(*HEAT Ponics *)
(*
	IF ((Modbus.Balkon_temp > Modbus.Balkon_set_temp+1)   ) THEN
		HW_balkon_heat		:= FALSE;
	END_IF

	IF ((Modbus.Balkon_temp <  Modbus.Balkon_set_temp-1 ) ) THEN
		HW_balkon_heat		:=	TRUE;
	END_IF
*)
(*
pwm_par_balkon.bInstantPWMUpdate:=0;
pwm_par_balkon.tPWMPeriod:=T#5800ms;
pwm_par_balkon.tTaskCycleTime:=T#5ms;

pi_par_balkon.bARWOnIPartOnly:=0;
pi_par_balkon.fKp:=40;
pi_par_balkon.fOutMaxLimit:=100;
pi_par_balkon.fOutMinLimit:=0;
pi_par_balkon.tCtrlCycleTime:=T#5ms;
pi_par_balkon.tTaskCycleTime:=T#5ms;
pi_par_balkon.tTn:=T#30m;

pi_balkon(fSetpointValue:=Modbus.Balkon_set_temp, fActualValue :=Modbus.Balkon_temp, fManSyncValue :=0, bSync:=0, eMode:=2,bHold:=0, stParams:=pi_par_balkon, fOut => );
pwm_balkon(fPwmInput:=pi_balkon.fOut, eMode:=2, stParams:=pwm_par_balkon, bPwmOutBitPos=>HW_balkon_heat );
*)
END_PROGRAM

(* POU ExtractTime, ST *)
FUNCTION_BLOCK ExtractTime
VAR_INPUT
	tm:TOD;
END_VAR
VAR_OUTPUT
	h, m	: UINT;
END_VAR
VAR
	tw	: DWORD;

END_VAR
tw:=TOD_TO_DWORD(tm);
tw:=tw/(1000*60);
m:=DWORD_TO_UINT(tw MOD 60);
h:=DWORD_TO_UINT(tw / 60);
END_FUNCTION_BLOCK

(* POU Thermocontrol, ST *)
PROGRAM Thermocontrol
VAR
(*	period_sec		: INT:=120;  *)  (* Частота работы термостата, секунды*)
	gisterezis		: REAL:=0.2; (*Гистерезис термостата, градусы цельсия *)
	Timer1			: TON;
	Timer1Q			: BOOL;
	state			: INT:=0;
	 tTimerValue		: TIME:=t#120s;  (* Частота работы термостата, секунды*)
	pi_1f, pi_2f, pi_sauna 			: FB_CTRL_PI;
	pwm_1f, pwm_2f, pwm_sauna1	: FB_CTRL_PWM_OUT;

	pi_balkon 			: FB_CTRL_PI;
	pwm_balkon			: FB_CTRL_PWM_OUT;

	pi_septik				: FB_CTRL_PI;
	pwm_septik			: FB_CTRL_PWM_OUT;
	Power_septik			: UINT:=75;


END_VAR
(* tTimerValue := DINT_TO_TIME(period_sec*1000); *)

pwm_par_1f.bInstantPWMUpdate:=0;
pwm_par_1f.tPWMPeriod:=T#5135ms;
pwm_par_1f.tTaskCycleTime:=T#10ms;

pwm_par_2f.bInstantPWMUpdate:=0;
pwm_par_2f.tPWMPeriod:=T#5735ms;
pwm_par_2f.tTaskCycleTime:=T#10ms;


pwm_par_balkon.bInstantPWMUpdate:=0;
pwm_par_balkon.tPWMPeriod:=T#5800ms;
pwm_par_balkon.tTaskCycleTime:=T#10ms;
pi_par_balkon.bARWOnIPartOnly:=0;
pi_par_balkon.fKp:=40;
pi_par_balkon.fOutMaxLimit:=100;
pi_par_balkon.fOutMinLimit:=0;
pi_par_balkon.tCtrlCycleTime:=T#10ms;
pi_par_balkon.tTaskCycleTime:=T#10ms;
pi_par_balkon.tTn:=T#30m;

IF Modbus.Heat_pipe_septik_winter = TRUE THEN
	pwm_par_septik.bInstantPWMUpdate:=0;
	pwm_par_septik.tPWMPeriod:=T#15000ms;
	pwm_par_septik.tTaskCycleTime:=T#10ms;
	pwm_septik(fPwmInput:=Power_septik, eMode:=2, stParams:=pwm_par_septik, bPwmOutBitPos=>HW_septik_heat );

END_IF

(*
pi_par_septik.bARWOnIPartOnly:=0;
pi_par_septik.fKp:=40;
pi_par_septik.fOutMaxLimit:=100;
pi_par_septik.fOutMinLimit:=0;
pi_par_septik.tCtrlCycleTime:=T#5ms;
pi_par_septik.tTaskCycleTime:=T#5ms;
pi_par_septik.tTn:=T#30m;
*)





pi_balkon(fSetpointValue:=Modbus.Balkon_set_temp, fActualValue :=Modbus.Balkon_temp, fManSyncValue :=0, bSync:=0, eMode:=2,bHold:=0, stParams:=pi_par_balkon, fOut => );
pwm_balkon(fPwmInput:=pi_balkon.fOut, eMode:=2, stParams:=pwm_par_balkon, bPwmOutBitPos=>HW_balkon_heat );




pwm_par_sauna.bInstantPWMUpdate:=0;
pwm_par_sauna.tPWMPeriod:=T#300s;
pwm_par_sauna.tTaskCycleTime:=T#5ms;


pi_par_1f.bARWOnIPartOnly:=0;
pi_par_1f.fKp:=40;
pi_par_1f.fOutMaxLimit:=100;
pi_par_1f.fOutMinLimit:=0;
pi_par_1f.tCtrlCycleTime:=T#5ms;
pi_par_1f.tTaskCycleTime:=T#5ms;
pi_par_1f.tTn:=T#30m;

pi_par_sauna.bARWOnIPartOnly:=0;
pi_par_sauna.fKp:=40;
pi_par_sauna.fOutMaxLimit:=100;
pi_par_sauna.fOutMinLimit:=0;
pi_par_sauna.tCtrlCycleTime:=T#5ms;
pi_par_sauna.tTaskCycleTime:=T#5ms;
pi_par_sauna.tTn:=T#30m;

(**)
	pi_1f(fSetpointValue:=Modbus.First_floor_temp_target, fActualValue :=INT_TO_REAL(HW_temp_first_floor)/10, fManSyncValue :=0, bSync:=0, eMode:=2,bHold:=0, stParams:=pi_par_1f, fOut => );
(*	pi_1f(fSetpointValue:=Modbus.First_floor_temp_target, fActualValue :=Internal.First_floor_temp_SHT30, fManSyncValue :=0, bSync:=0, eMode:=2,bHold:=0, stParams:=pi_par_1f, fOut => );*)

	pwm_1f(fPwmInput:=pi_1f.fOut, eMode:=2, stParams:=pwm_par_1f, bPwmOutBitPos=>HW_heat_first_floor );

	pi_2f(fSetpointValue:=Modbus.Second_floor_temp_target, fActualValue :=INT_TO_REAL(HW_temp_second_floor)/10, fManSyncValue :=0, bSync:=0, eMode:=2,bHold:=0, stParams:=pi_par_1f, fOut => );
	pwm_2f(fPwmInput:=pi_2f.fOut, eMode:=2, stParams:=pwm_par_2f, bPwmOutBitPos=>HW_heat_second_floor );

(* SAUNA PID*)
(*
	pi_sauna(fSetpointValue:=Modbus.Sauna_temp_target, fActualValue :=INT_TO_REAL(HW_temp_sauna)/10, fManSyncValue :=0, bSync:=0, eMode:=2,bHold:=0, stParams:=pi_par_sauna, fOut => );
	pwm_sauna1(fPwmInput:=pi_sauna.fOut, eMode:=2, stParams:=pwm_par_sauna, bPwmOutBitPos=>HW_heat_Sauna );
*)

CASE state OF
0:
(*	IF (Modbus.First_floor_temp > Modbus.First_floor_temp_target+gisterezis ) THEN
		HW_heat_first_floor:=FALSE;
	END_IF

	IF ((Modbus.First_floor_temp <  Modbus.First_floor_temp_target-gisterezis) AND (Modbus.First_floor_temp <>0)  ) THEN
		HW_heat_first_floor:=TRUE;
	END_IF
*)

	state:=1;

1:
(*	IF (Modbus.Second_floor_temp > Modbus.Second_floor_temp_target+gisterezis ) THEN
		HW_heat_Second_floor:=FALSE;
	END_IF

	IF ((Modbus.Second_floor_temp <  Modbus.Second_floor_temp_target-gisterezis ) AND (Modbus.Second_floor_temp <>0)) THEN
		HW_heat_Second_floor:=TRUE;
	END_IF
*)
	state:=2;
2:
(* SAUNA GISTEREZIS *)

	IF (Modbus.Sauna_temp > Modbus.Sauna_temp_target+gisterezis ) THEN
		HW_heat_Sauna:=FALSE;
	END_IF

	IF ((Modbus.Sauna_temp <  Modbus.Sauna_temp_target-gisterezis ) AND (Modbus.Sauna_temp <>0)) THEN
		HW_heat_Sauna:=TRUE;
	END_IF
	state:=3;
3:


IF (Modbus.Sport_temp > Modbus.Sport_temp_target+gisterezis OR HW_heat_Sauna=TRUE ) THEN
		HW_heat_sport:=FALSE;
	END_IF

	IF ((Modbus.Sport_temp <  Modbus.Sport_temp_target-gisterezis ) AND (Modbus.Sport_temp <>0)  AND HW_heat_Sauna=FALSE) THEN
		HW_heat_sport:=TRUE;
	END_IF



	state:=4;

4:
	IF (Modbus.Underfloor_temp > Modbus.Underfloor_temp_target+gisterezis AND Modbus.Underfloor_hum < Modbus.Underfloor_humidity_target-1 ) THEN
		HW_heat_underfloor:=FALSE;
	END_IF

	IF ((Modbus.Underfloor_temp <  Modbus.Underfloor_temp_target-gisterezis OR Modbus.Underfloor_hum > Modbus.Underfloor_humidity_target+1) AND (Modbus.Underfloor_temp <>0)) THEN
		HW_heat_Underfloor:=TRUE;
	END_IF

	state:=100;



100:


	Timer1(IN:=NOT Timer1Q , PT:=tTimerValue , Q=>Timer1Q , ET=> );
		IF timer1.q THEN

		state:=0;
		END_IF



END_CASE
END_PROGRAM

(* POU Sensors, ST *)
PROGRAM Sensors
VAR
(*	Period_sensors_read		: INT:=30; *) (* Частота присвоения значений аналоговых температурных датчиков с модулей KL, секунды *)
	Timer					: TON;
	TimerQ					: BOOL;
	tTimerValue				: TIME:=t#30s; (* Частота присвоения значений аналоговых температурных датчиков с модулей KL, секунды *)
	Trigger_water_cold: F_TRIG;
	Water_count_house		: REAL;
	Water_count_teplica		: REAL;
END_VAR
Timer();
Trigger_water_cnt_impulse_teplica(CLK:=HW_I_rez5);

Trigger_water_cold(CLK :=HW_water_counter);
IF (Trigger_water_cold.Q) THEN

	(*Modbus.Kitchen_stat_cold_water:=Modbus.Kitchen_stat_cold_water+1; *)
	Water_count_house	:=	Water_count_house+1;
	Modbus.Sensor_house_water_imp	:=	Modbus.Sensor_house_water_imp+1;
END_IF

IF Trigger_water_cnt_impulse_teplica.Q THEN
	Water_count_teplica	:=	Water_count_teplica+1;
	Modbus.Teplica_cnt_water_pipe	:= 	Modbus.Teplica_cnt_water_pipe+1;
END_IF




(* tTimerValue := DINT_TO_TIME(Period_sensors_read*1000); *)

	Timer(IN:=NOT TimerQ , PT:=tTimerValue , Q=>TimerQ , ET=> );
	IF timer.q THEN

		Modbus.First_floor_temp		:=	INT_TO_REAL(HW_temp_first_floor)/10;
(*		Modbus.First_floor_temp		:=	Internal.First_floor_temp_SHT30; *)

		Modbus.Second_floor_temp	:=	INT_TO_REAL(HW_temp_second_floor)/10;
		Modbus.Sauna_temp			:=	INT_TO_REAL(HW_temp_sauna)/10;
		Modbus.Sport_temp			:=	INT_TO_REAL(HW_temp_sport)/10;

		Modbus.Underfloor_temp		:=	INT_TO_REAL(HW_temp_underfloor)/10;
(*		Modbus.Sport_underfloor_temp	:=	INT_TO_REAL(HW_temp_sport_underfloor)/10;	*)
		Modbus.Street_temp			:=	INT_TO_REAL(HW_temp_street)/10;
		Modbus.Vent_temp			:=	INT_TO_REAL(HW_temp_vent)/10;

		Modbus.Balkon_temp			:=	INT_TO_REAL(HW_temp_balkon)/10;
(*		Modbus.Drovnik_temp			:=	INT_TO_REAL(HW_temp_drovnik)/10;
		Modbus.Sklad_temp			:= 	INT_TO_REAL(HW_temp_sklad)/10;	*)

	END_IF
END_PROGRAM

(* POU Security_new, ST *)
PROGRAM Security_new
VAR
(*	TRIG_PIR_terrasa			:	F_TRIG;
	TRIG_PIR_zapad			:	F_TRIG;
	TRIG_PIR_vostok			:	F_TRIG;
	TRIG_PIR_sport			:	F_TRIG;
	TRIG_GERKON_drovnik	:	F_TRIG;
	TRIG_sensor_smoke_1floor:	F_TRIG;

	trig_mem_terrasa				:	BOOL:=FALSE;
	trig_mem_zapad				:	BOOL:=FALSE;
	trig_mem_vostok				:	BOOL:=FALSE;
	trig_mem_sport				:	BOOL:=FALSE;
	trig_mem_drovnik				:	BOOL:=FALSE;
	trig_mem_sensor_smoke_1floor	:	BOOL:=FALSE;
*)
END_VAR
iobroker.PIR_terrasa			 :=HW_PIR_terrasa;
iobroker.PIR_zapad			 :=HW_PIR_zapad;
iobroker.PIR_vostok 			 :=HW_PIR_vostok;
iobroker.PIR_sport			 :=HW_PIR_sport;
iobroker.GERKON_drovnik		 :=HW_GERKON_drovnik;
(*
Modbus.Smoke_1floor				 :=HW_sensor_smoke_1floor;
Modbus.Smoke_2floor			 	:=HW_sensor_smoke_2floor;
Modbus.Smoke_sport				 :=HW_sensor_smoke_sport;
Modbus.Smoke_sklad				 :=HW_sensor_smoke_sklad;
Modbus.Smoke_drovnik			 :=HW_sensor_smoke_drovnik;
*)

Modbus.PIR_terrasa			 :=HW_PIR_terrasa;
Modbus.PIR_zapad			 :=HW_PIR_zapad;
Modbus.PIR_vostok 			 :=HW_PIR_vostok;
Modbus.PIR_sport				 :=HW_PIR_sport;
Modbus.PIR_north_zapad		 :=HW_PIR_north_zapad;
Modbus.PIR_north_vostok		 :=HW_PIR_north_vostok;

Modbus.GERKON_door		 :=HW_GERKON_door;
Modbus.GERKON_drovnik		 :=HW_GERKON_drovnik;
Modbus.GERKON_sklad		 :=HW_GERKON_sklad;



(* Modbus.Smoke				 :=HW_sensor_smoke_1floor; *)
END_PROGRAM

(* POU RS485read, ST *)
PROGRAM RS485read
VAR

	tTimerValue				: TIME	:=	t#60s; (* Период опроса RS485*)
	FtrigBusy				: F_TRIG;
	timeoutvalue				: TIME := T#2000ms;		(* timeout while waiting for an answer of the modbus slave *)
	state					: INT;
	busy					: BOOL;
	LastErrorstate				: INT;
	LastModbusError			: ST_ModbusErrorDiagnostics;
	CounterError				: DINT;
	CounterSuccess			: DINT;
	i,k,l						: INT:=1;

	teplica_ADM4188_id			: BYTE:=16#45;
	klubnika_WP8025ADAM		: BYTE:=16#46;
	klubnika_SHT30				: BYTE:=16#64;


	sensors_SHT20_v1_id			: ARRAY[1..3] OF BYTE:= 16#0F, 16#05, 16#36;
	sensors_SHT20_v1_hum		: ARRAY[1..3] OF REAL:=3(0);
	sensors_SHT20_v1_temp		: ARRAY[1..3] OF REAL:=3(0);

(*	sensors_SHT20_v2_id			: ARRAY[1..1] OF BYTE:=  16#0A; *)
	sensors_SHT20_v2_id			: ARRAY[1..1] OF BYTE:=  16#35;

	sensors_SHT20_v2_hum		: ARRAY[1..1] OF REAL:=1(0);
	sensors_SHT20_v2_temp		: ARRAY[1..1] OF REAL:=1(0);


	sensors_SHT30_v3_id			: ARRAY[1..8] OF BYTE:= 16#14, 16#11,16#29, 16#30,16#07,16#08, 16#32, 16#35;
	sensors_SHT30_v3_hum		: ARRAY[1..8] OF REAL:=8(0);
	sensors_SHT30_v3_temp		: ARRAY[1..8] OF REAL:=8(0);

	sensors_CO2_id				: ARRAY[1..4] OF BYTE:=16#68, 16#69,16#6A, 16#6B ;
	sensors_CO2_ppm			: ARRAY[1..4] OF INT;

	house_DS18B20_id			: BYTE:=16#64;
	sensors_DS18B20_temp		: ARRAY[1..8] OF REAL:=8(0);
	parnik_DS18B20_id			: BYTE:=16#64;
	teplica_DS18B20_temp		: ARRAY[1..8] OF REAL:=8(0);
	teplica_gate_pt1000_id			: BYTE:=70;
	MBdata8_pt1000				 : ARRAY [1..8] OF INT;
	MBdata_teplica_gate_pt1000	: ARRAY [1..8] OF REAL;

	MBdata						 : ARRAY [1..2] OF INT;
	MBdata8						 : ARRAY [1..8] OF UINT;
	MBdata8_h					 : ARRAY [1..8] OF UINT;

	sensor_ponics_PH_id			: BYTE:= 16#4F ;
	sensor_teplica_PH_id			: BYTE:= 16#78 ;
	MBdata_sensor_ponics_PH	: ARRAY [1..4] OF INT;
	MBdata_sensor_teplica_PH	: ARRAY [1..4] OF INT;

	Teplica_tank_level_id			: BYTE:=1;
	Teplica_tankA_level_id		: BYTE:=2;
	Teplica_tankB_level_id		: BYTE:=3;

	Teplica_ph_sensor_low		: REAL;
	Teplica_ph_sensor_temp		: REAL;
	Teplica_ph_sensor_mv		: REAL;
(*	Teplica_temp_air				: REAL; *)
	Teplica_temp_pip_heat_in		: REAL;

	Ponics_ph_sensor_mv			: REAL;

	sensor_teplica_EC_id			: BYTE:= 16#C8 ;
	sensor_ponics_EC_id			: BYTE:= 16#51 ;
	sensor_ponics_EC2_id			: BYTE:= 16#50 ;
	sensor_ponics_EC_int			: INT;
	sensor_ponics_EC2_int		: INT;
	MBdata_sensor_teplica_EC		 : ARRAY [1..4] OF INT;
	MBdata_sensor_ponics_EC2	 :  INT;

	balkon_light_sensor_id			: BYTE:=16#5A;
	balkon_light_word2			: WORD;
	teplica_light_sensor_id			: BYTE:=16#3C;
	teplica_light_low				: WORD;
	teplica_light_high				: WORD;
	teplica_light_dword			: DWORD;
	teplica_light_array				: ARRAY [1..2] OF WORD;

	password_1				: ARRAY [1..6] OF BYTE:=6(1); (* пароль к меркуриям, по умолчанию 6 единиц*)
	crctest					: WORD;
	get_energy_E_T1			: FB_GET_ENERGY;
	get_energy_E_T2			: FB_GET_ENERGY;
	get_energy_MT			: FB_GET_ENERGY;
	get_supply				: FB_GET_SUPPLY;
	get_current				: FB_GET_CURRENT;
	get_power				: FB_GET_POWER;
	energyMT					: ARRAY[1..12,1..2] OF REAL;
	get_current_done			: BOOL;
	get_power_done			: BOOL;
	get_energy_E_T1_done	: BOOL;
	get_energy_E_T2_done	: BOOL;
	get_energy_MT_done		: BOOL;
	get_supply_done			: BOOL;
	arrReceive				: ARRAY[1..5] OF BYTE;
	arrSend					: ARRAY[1..5] OF BYTE;
	t,m, tr, none				: INT:=1;
	 e_rs1					: INT:=0;
	ponics_EC2_1				: REAL;
	ponics_EC2_2				: REAL;
	ponics_EC2_3				: REAL;
	ponics_EC2_4				: REAL;
	Modbus_errors			:DWORD;
	Modbus_array_errors		:ARRAY[0..254] OF BYTE;
	Balkon_CO2				: INT;
	Teplica_CO2				: INT;
	Timer_wait_RS			: TON;
	 tTimerValue_wait_RS1		: TIME:=t#2s;  (* *)
	cnt_err_read_tank			:UDINT;
	cnt_err_read_all			:UDINT;
	Temp_water_tank_DS		: REAL;
	Teplica_temp_panel		: REAL;
	teplica_tank_level_word	: ARRAY[0..17] OF WORD;
	teplica_tankA_level_word	: ARRAY[0..17] OF WORD;
	teplica_tankB_level_word	: ARRAY[0..17] OF WORD;

	Teplica_tank_level		: REAL;
	Teplica_tankA_level		: REAL;
	Teplica_tankB_level		: REAL;

	cnt_clear_di_2: BOOL;
	zero						: INT:=0;
	MBdataDI		 			 : ARRAY [1..8] OF UINT;
	Teplica_DO1			:	BOOL;
	Teplica_DO2			:	BOOL;
	Teplica_DO3			:	BOOL;
	Teplica_DO4			:	BOOL;
	Teplica_DO5			:	BOOL;
	Teplica_DO6			:	BOOL;
	Teplica_DO7			:	BOOL;
	Teplica_DO8			:	BOOL;

	MBdataDO_byte: BYTE;
	MBdataDO_byte_read: BYTE;
	test: BOOL;
END_VAR
(*Modbus.RS485_1_cnt_error		:= Modbus.RS485_1_cnt_error;
Modbus.RS485_1_cnt_success	:= Modbus.RS485_1_cnt_success;
*)

MBdataDO_byte.0			:=	Modbus.Teplica_pomp_fertA;
MBdataDO_byte.1			:=	Modbus.Teplica_pomp_fertB;
MBdataDO_byte.2			:=	Modbus.Teplica_zone_poliv;
MBdataDO_byte.3			:=	Modbus.Teplica_window_opener;
MBdataDO_byte.4			:=	Modbus.Teplica_pomp_cold;
MBdataDO_byte.5			:=	Modbus.Teplica_tank_heat;
MBdataDO_byte.7			:= 	Modbus.Light_garden;

CASE state OF
0:
		MB.ReadRegs(Execute:= FALSE);
		state := 2;

		e_rs1	:=0;
		Modbus_array_errors[0] :=0;
		Modbus_array_errors[1] :=0;
		Modbus_array_errors[2] :=0;
		Modbus_array_errors[3] :=0;
		Modbus_array_errors[4] :=0;
		Modbus_array_errors[5] :=0;
		Modbus_array_errors[6] :=0;
		Modbus_array_errors[7] :=0;
		Modbus_array_errors[8] :=0;
		Modbus_array_errors[9] :=0;
		Modbus_array_errors[10] :=0;



1:

		MB.ReadInputRegs(
			UnitID:= sensors_SHT20_v2_id[l],
			Quantity:= 2,
			MBAddr:= 512,
			cbLength:= 4,
			pMemoryAddr:= ADR(MBdata),
			Execute:= TRUE,
			Timeout:= timeoutvalue,
			Busy => busy,
		);
		IF NOT busy THEN
			IF (mb.Error = FALSE ) THEN
				sensors_SHT20_v2_temp[l]:=INT_TO_REAL(MBdata[1])/10;
				sensors_SHT20_v2_hum[l]:=INT_TO_REAL(MBdata[2])/10;
			ELSE
				Modbus_array_errors[e_rs1]	:= sensors_SHT20_v2_id[l];
				e_rs1	:= e_rs1+1;
			END_IF

			l:=l+1;
			MB.ReadRegs(Execute:= FALSE);
			IF (l>1 )	THEN
				l:=1;
				Modbus.Balkon_hum	:=	sensors_SHT20_v2_hum[1];

(*				Internal.Sport_underfloor_temp_SHT20		:=	sensors_SHT20_v2_temp[1];
				Internal.Sport_underfloor_hum				:=	sensors_SHT20_v2_hum[1];


				Modbus.Sport_underfloor_temp_SHT20		:=	(sensors_SHT20_v2_temp[1]);
				Modbus.Sport_underfloor_hum				:=	(sensors_SHT20_v2_hum[1]);
*)
				state :=2;
			ELSE
				state :=1;
			END_IF

		END_IF



2:
		MB.ReadRegs(
			UnitID:= sensors_SHT20_v1_id[i],
			Quantity:= 2,
			MBAddr:= 0,
			cbLength:= 4,
			pMemoryAddr:= ADR(MBdata),
			Execute:= TRUE,
			Timeout:= timeoutvalue,
			Busy => busy,
		);
		IF NOT busy THEN
			IF (mb.Error = FALSE ) THEN
				sensors_SHT20_v1_temp[i]:=INT_TO_REAL(MBdata[1])/10;
				sensors_SHT20_v1_hum[i]:=INT_TO_REAL(MBdata[2])/10;
			ELSE
				Modbus_array_errors[e_rs1]	:= sensors_SHT20_v1_id[i];

				e_rs1	:= e_rs1+1;
			END_IF
			i:=i+1;
			MB.ReadRegs(Execute:= FALSE);
			IF (i>3 )	THEN
				i:=1;
				Internal.Street_temp_SHT20			:=	sensors_SHT20_v1_temp[1];
				Internal.Street_hum				:=	sensors_SHT20_v1_hum[1];
				Internal.Sklad_temp_SHT20			:=	sensors_SHT20_v1_temp[2];
				Internal.Sklad_hum				:=	sensors_SHT20_v1_hum[2];

				Modbus.Street_temp_SHT20		:=	sensors_SHT20_v1_temp[1];
				Modbus.Street_hum				:=	sensors_SHT20_v1_hum[1];
				Modbus.Sklad_temp_SHT20		:=	sensors_SHT20_v1_temp[2];
				Modbus.Sklad_hum				:=	sensors_SHT20_v1_hum[2];
				Modbus.Parnik_sht_air_temp		:=	(sensors_SHT20_v1_temp[3])/10;
				Modbus.Parnik_sht_air_hum		:=	(sensors_SHT20_v1_hum[3])/10;
				state :=3;
			ELSE
				state :=2;
			END_IF

		END_IF


3:
		MB.ReadRegs(
			UnitID:= sensors_SHT30_v3_id[i],
			Quantity:= 2,
			MBAddr:= 512,
			cbLength:= 4,
			pMemoryAddr:= ADR(MBdata),
			Execute:= TRUE,
			Timeout:= timeoutvalue,
			Busy => busy,
		);
		IF NOT busy THEN
			IF (mb.Error = FALSE ) THEN
				sensors_SHT30_v3_temp[i]:=INT_TO_REAL(MBdata[1])/10;
				sensors_SHT30_v3_hum[i]:=INT_TO_REAL(MBdata[2])/10;
			ELSE
				Modbus_array_errors[e_rs1]	:= sensors_SHT30_v3_id[i];

				e_rs1	:= e_rs1+1;
			END_IF
			i:=i+1;
			MB.ReadRegs(Execute:= FALSE);
			IF (i>8 )	THEN
				i:=1;
				Internal.Drovnik_temp_SHT30		:=	sensors_SHT30_v3_temp[1];
				Internal.Drovnik_hum				:=	sensors_SHT30_v3_hum[1];
				Internal.Sport_temp_SHT30			:=	sensors_SHT30_v3_temp[2];
				Internal.Sport_hum					:=	sensors_SHT30_v3_hum[2];
				Internal.First_floor_temp_SHT30		:=	sensors_SHT30_v3_temp[3];
				Internal.First_floor_hum				:=	sensors_SHT30_v3_hum[3];
				Internal.Second_floor_temp_SHT30	:=	sensors_SHT30_v3_temp[4];
				Internal.Second_floor_hum			:=	sensors_SHT30_v3_hum[4];
				Internal.Underfloor_temp_SHT30		:=	sensors_SHT30_v3_temp[5];
				Internal.Underfloor_hum			:=	sensors_SHT30_v3_hum[5];
				Internal.Sport_underfloor_temp_SHT30		:=	sensors_SHT30_v3_temp[6];
				Internal.Sport_underfloor_hum				:=	sensors_SHT30_v3_hum[6];
				Internal.Teplica_temp_SHT30		:=	sensors_SHT30_v3_temp[7];
				Internal.Teplica_hum_SHT30		:=	sensors_SHT30_v3_hum[7];

				Modbus.Drovnik_temp_SHT30		:=	sensors_SHT30_v3_temp[1];
				Modbus.Drovnik_hum				:=	sensors_SHT30_v3_hum[1];
				Modbus.Sport_temp_SHT30		:=	sensors_SHT30_v3_temp[2];
				Modbus.Sport_hum				:=	sensors_SHT30_v3_hum[2];
				Modbus.First_floor_temp_SHT30	:=	sensors_SHT30_v3_temp[3];
				Modbus.First_floor_hum			:=	sensors_SHT30_v3_hum[3];
				Modbus.Second_floor_temp_SHT30	:=	sensors_SHT30_v3_temp[4];
				Modbus.Second_floor_hum			:=	sensors_SHT30_v3_hum[4];
				Modbus.Underfloor_temp_SHT30	:=	sensors_SHT30_v3_temp[5];
				Modbus.Underfloor_hum			:=	sensors_SHT30_v3_hum[5];
				Modbus.Sport_underfloor_temp_SHT30		:=	(sensors_SHT30_v3_temp[6]);
				Modbus.Sport_underfloor_hum				:=	(sensors_SHT30_v3_hum[6]);
				Modbus.Teplica_temp_SHT30		:=	sensors_SHT30_v3_temp[7];
				Modbus.Teplica_temp_air			:=	sensors_SHT30_v3_temp[7];
				Modbus.Teplica_hum_SHT30		:=	sensors_SHT30_v3_hum[7];
				Modbus.Balkon_hum				:=	sensors_SHT30_v3_hum[8];
				state :=4;
			ELSE
				state :=3;
			END_IF

		END_IF

4:
		MB.ReadInputRegs(
			UnitID:=sensors_CO2_id[k], (* station address *)
			Quantity:= 1,
			MBAddr:= 3,
			cbLength:= 2,
			pMemoryAddr:= ADR(MBdata),
			Execute:= TRUE,
			Timeout:= timeoutvalue,
			Busy => busy	);
		IF NOT busy THEN
			IF (mb.Error = FALSE ) THEN
				sensors_CO2_ppm[k]	:=	(MBdata[1]);
			ELSE
				Modbus_array_errors[e_rs1]	:= sensors_CO2_id[k];
				e_rs1	:= e_rs1+1;
			END_IF
			k:=k+1;
			MB.ReadRegs(Execute:= FALSE);
			IF (k>4 )	THEN
				k:=1;
				Modbus.Second_floor_CO2		:=	(sensors_CO2_ppm[1]);
				Modbus.First_floor_CO2		:=	(sensors_CO2_ppm[2]);
				Modbus.Balkon_CO2			:=	(sensors_CO2_ppm[3]);
				Modbus.Teplica_CO2			:=	(sensors_CO2_ppm[4]);

				state :=6;
			ELSE
				state :=4;
			END_IF
		END_IF




5:

		MB.ReadRegs(
			UnitID:= house_DS18B20_id,
			Quantity:= 8,
			MBAddr:= 0,
			cbLength:= 16,
			pMemoryAddr:= ADR(MBdata8_h),
			Execute:= TRUE,
			Timeout:= timeoutvalue,
			Busy => busy,
		);
		IF NOT busy THEN
			IF (mb.Error = FALSE ) THEN
(*				sensors_DS18B20_temp[1]:=INT_TO_REAL(MBdata8_h[1])/10;
				sensors_DS18B20_temp[2]:=INT_TO_REAL(MBdata8_h[2])/10;
				sensors_DS18B20_temp[3]:=INT_TO_REAL(MBdata8_h[3])/10;
				sensors_DS18B20_temp[4]:=INT_TO_REAL(MBdata8_h[4])/10;
*)
				IF (MBdata8_h[1] < 10000)
					THEN	sensors_DS18B20_temp[1]:=UINT_TO_REAL(MBdata8_h[1])/10;
				ELSE
					sensors_DS18B20_temp[1]:=-1*UINT_TO_REAL(MBdata8_h[1]-10000)/10;
				END_IF

				IF (MBdata8_h[2] < 10000)
					THEN	sensors_DS18B20_temp[2]:=UINT_TO_REAL(MBdata8_h[2])/10;
				ELSE
					sensors_DS18B20_temp[2]:=-1*UINT_TO_REAL(MBdata8_h[2]-10000)/10;
				END_IF


				IF (MBdata8_h[3] < 10000)
					THEN	sensors_DS18B20_temp[3]:=UINT_TO_REAL(MBdata8_h[3])/10;
				ELSE
					sensors_DS18B20_temp[3]:=-1*UINT_TO_REAL(MBdata8_h[3]-10000)/10;
				END_IF

				IF (MBdata8_h[5] < 10000)
					THEN	sensors_DS18B20_temp[5]:=UINT_TO_REAL(MBdata8_h[5])/10;
				ELSE
					sensors_DS18B20_temp[5]:=-1*UINT_TO_REAL(MBdata8_h[5]-10000)/10;
				END_IF



				IF  (sensors_DS18B20_temp[5] <>0 AND sensors_DS18B20_temp[5] <>85)	THEN
					Modbus.Rezerv_temp			:=	sensors_DS18B20_temp[5];
				END_IF
(*
				IF  (sensors_DS18B20_temp[2] <>0 AND sensors_DS18B20_temp[2] <>85)	THEN
					Modbus.		:=	sensors_DS18B20_temp[2];
				END_IF

				IF  (sensors_DS18B20_temp[3] <>0 AND sensors_DS18B20_temp[3] <>85)	THEN
					Modbus. 	:=	sensors_DS18B20_temp[3];
				END_IF

				IF  (sensors_DS18B20_temp[4] <>0 AND sensors_DS18B20_temp[4] <>85)	THEN
					Modbus. 	:=	sensors_DS18B20_temp[4];
				END_IF
*)

			ELSE
				Modbus_array_errors[e_rs1]	:= house_DS18B20_id;
				e_rs1	:= e_rs1+1;
			END_IF
			MB.ReadRegs(Execute:= FALSE);
			state:=6;

		END_IF


6:

		MB.ReadRegs(
			UnitID:= parnik_DS18B20_id,
			Quantity:= 8,
			MBAddr:= 0,
			cbLength:= 16,
			pMemoryAddr:= ADR(MBdata8),
			Execute:= TRUE,
			Timeout:=  T#2000ms,
			Busy => busy,
		);
		IF NOT busy THEN
			IF (MB.Error = FALSE ) THEN
				IF (MBdata8[1] < 10000)
					THEN	teplica_DS18B20_temp[1]:=UINT_TO_REAL(MBdata8[1])/10;
				ELSE
					teplica_DS18B20_temp[1]:=-1*UINT_TO_REAL(MBdata8[1]-10000)/10;
				END_IF

				IF (MBdata8[2] < 10000)
					THEN	teplica_DS18B20_temp[2]:=UINT_TO_REAL(MBdata8[2])/10;
				ELSE
					teplica_DS18B20_temp[2]:=-1*UINT_TO_REAL(MBdata8[2]-10000)/10;
				END_IF


				IF (MBdata8[3] < 10000)
					THEN	teplica_DS18B20_temp[3]:=UINT_TO_REAL(MBdata8[3])/10;
				ELSE
					teplica_DS18B20_temp[3]:=-1*UINT_TO_REAL(MBdata8[3]-10000)/10;
				END_IF

				IF (MBdata8[4] < 10000)
					THEN	teplica_DS18B20_temp[4]:=UINT_TO_REAL(MBdata8[4])/10;
				ELSE
					teplica_DS18B20_temp[4]:=-1*UINT_TO_REAL(MBdata8[4]-10000)/10;
				END_IF

				IF (MBdata8[5] < 10000)
					THEN	teplica_DS18B20_temp[5]:=UINT_TO_REAL(MBdata8[5])/10;
				ELSE
					teplica_DS18B20_temp[5]:=-1*UINT_TO_REAL(MBdata8[5]-10000)/10;
				END_IF


				IF  (teplica_DS18B20_temp[1] <>0 AND teplica_DS18B20_temp[1] <>85 AND teplica_DS18B20_temp[1] > -60  )	THEN
					Modbus.Parnik_air_temp	:= 		teplica_DS18B20_temp[1];
				END_IF

				IF  (teplica_DS18B20_temp[2] <>0 AND teplica_DS18B20_temp[2] <>85 AND teplica_DS18B20_temp[2] > -60)	THEN
					Modbus.Parnik_ground_temp		:=	teplica_DS18B20_temp[2];
				END_IF


				IF  (teplica_DS18B20_temp[3] <>0 AND teplica_DS18B20_temp[3] <>85  AND teplica_DS18B20_temp[3] > -60)	THEN
					Modbus.Parnik_pipe_temp	 	:=	teplica_DS18B20_temp[3];
				END_IF

(*				IF  (teplica_DS18B20_temp[4] <>0 AND teplica_DS18B20_temp[4] <>85 AND teplica_DS18B20_temp[4] > -60)	THEN

					Temp_water_tank_DS				:=	teplica_DS18B20_temp[4];
				END_IF

				IF  (teplica_DS18B20_temp[5] <>0 AND teplica_DS18B20_temp[5] <>85 AND teplica_DS18B20_temp[5] > -60)	THEN
					Teplica_temp_pip_heat_in 	:=	teplica_DS18B20_temp[5];
				END_IF

				IF  (teplica_DS18B20_temp[1]  = 0 OR teplica_DS18B20_temp[2]  = 0 OR teplica_DS18B20_temp[3]  = 0 OR teplica_DS18B20_temp[4]  = 0OR  teplica_DS18B20_temp[5]  = 0) THEN
					cnt_err_read_all	:=	cnt_err_read_all+1;
				END_IF

*)


			ELSE
				Modbus_array_errors[e_rs1]	:= parnik_DS18B20_id;
				e_rs1	:= e_rs1+1;
			END_IF
			MB.ReadRegs(Execute:= FALSE);
				state:=7;

		END_IF




7:

		MB.ReadRegs(
			UnitID:= balkon_light_sensor_id,
			Quantity:= 1,
			MBAddr:= 6,
			cbLength:= 2,
			pMemoryAddr:= ADR(balkon_light_word2),
			Execute:= TRUE,
			Timeout:= timeoutvalue,
			Busy => busy,
		);
		IF NOT busy THEN
			IF (mb.Error = FALSE ) THEN
				Modbus.Balkon_light_lux		:=	WORD_TO_UDINT(balkon_light_word2);
			ELSE
				Modbus_array_errors[e_rs1]	:= balkon_light_sensor_id;
				e_rs1	:= e_rs1+1;
			END_IF
			MB.ReadRegs(Execute:= FALSE);
			state:=8;
		END_IF

8:

		MB.ReadRegs(
			UnitID:= teplica_light_sensor_id,
			Quantity:= 2,
			MBAddr:= 2,
			cbLength:= 4,
			pMemoryAddr:= ADR(teplica_light_array),
			Execute:= TRUE,
			Timeout:= timeoutvalue,
			Busy => busy,
		);
		IF NOT busy THEN
			IF (MB.Error = FALSE ) THEN
				teplica_light_high:=teplica_light_array[1];
				teplica_light_low:=teplica_light_array[2];
				teplica_light_dword:=(teplica_light_array[1]*65535)+teplica_light_array[2];
				Modbus.Teplica_light_lux		:=	DWORD_TO_REAL(teplica_light_dword);


			ELSE
				Modbus_array_errors[e_rs1]	:= teplica_light_sensor_id;
				e_rs1	:= e_rs1+1;
			END_IF
			MB.ReadRegs(Execute:= FALSE);
			state:=9;
		END_IF

9:

		MB.ReadRegs(
			UnitID:= sensor_ponics_PH_id,
			Quantity:= 4,
			MBAddr:= 0,
			cbLength:= 8,
			pMemoryAddr:= ADR(MBdata_sensor_ponics_PH),
			Execute:= TRUE,
			Timeout:= timeoutvalue,
			Busy => busy,
		);
		IF NOT busy THEN
			IF (mb.Error = FALSE ) THEN
				Modbus.Ponics_PH			:=	INT_TO_REAL(MBdata_sensor_ponics_PH[1])/100;
				Modbus.Ponics_tank_temp		:=	INT_TO_REAL(MBdata_sensor_ponics_PH[3])/10;
				Ponics_ph_sensor_mv			:=	INT_TO_REAL(MBdata_sensor_ponics_PH[4]);

			ELSE
				Modbus_array_errors[e_rs1]	:= sensor_ponics_PH_id;
				e_rs1	:= e_rs1+1;

			END_IF
			MB.ReadRegs(Execute:= FALSE);
			state:=11;
		END_IF

10:

		MB.ReadRegs(
			UnitID:= sensor_teplica_PH_id,
			Quantity:= 4,
			MBAddr:= 0,
			cbLength:= 8,
			pMemoryAddr:= ADR(MBdata_sensor_teplica_PH),
			Execute:= TRUE,
			Timeout:= timeoutvalue,
			Busy => busy,
		);
		IF NOT busy THEN
			IF (MB.Error = FALSE ) THEN
				Modbus.Teplica_sensor_soil_PH	:=	INT_TO_REAL(MBdata_sensor_teplica_PH[1])/100;
				Teplica_ph_sensor_low			:=	INT_TO_REAL(MBdata_sensor_teplica_PH[2])/10;
				Teplica_ph_sensor_temp			:=	INT_TO_REAL(MBdata_sensor_teplica_PH[3])/10;
				Teplica_ph_sensor_mv			:=	INT_TO_REAL(MBdata_sensor_teplica_PH[4]);

			ELSE
				Modbus_array_errors[e_rs1]	:= sensor_teplica_PH_id;
				e_rs1	:= e_rs1+1;

			END_IF
			MB.ReadRegs(Execute:= FALSE);
			state:=11;
		END_IF


11:

		MB.ReadRegs(
			UnitID:= sensor_ponics_EC_id,
			Quantity:= 1,
			MBAddr:= 2,
			cbLength:= 2,
			pMemoryAddr:= ADR(sensor_ponics_EC_int),
			Execute:= TRUE,
			Timeout:= timeoutvalue,
			Busy => busy,
		);
		IF NOT busy THEN
			IF (mb.Error = FALSE ) THEN
			Modbus.Ponics_EC	:=	 INT_TO_REAL(sensor_ponics_EC_int)/1000;
				IF(Modbus.Ponics_EC < 0)	THEN
					Modbus.Ponics_EC	:= 0;
				END_IF
			ELSE
				Modbus_array_errors[e_rs1]	:= sensor_ponics_EC_id;
				e_rs1	:= e_rs1+1;
			END_IF
			MB.ReadRegs(Execute:= FALSE);
			state:=12;
		END_IF

12:

		MB.ReadRegs(
			UnitID:= sensor_teplica_EC_id,
			Quantity:= 4,
			MBAddr:= 0,
			cbLength:= 8,
			pMemoryAddr:= ADR(MBdata_sensor_teplica_EC),
			Execute:= TRUE,
			Timeout:= timeoutvalue,
			Busy => busy,
		);
		IF NOT busy THEN
			IF (MB.Error = FALSE ) THEN
			Modbus.Teplica_sensor_soil_Hum	:=	INT_TO_REAL(MBdata_sensor_teplica_EC[1])/10;
			Modbus.Teplica_sensor_soil_Temp	:=	INT_TO_REAL(MBdata_sensor_teplica_EC[2])/10;
			Modbus.Teplica_sensor_soil_EC	:=	INT_TO_REAL(MBdata_sensor_teplica_EC[3])/1000;
			Modbus.Teplica_sensor_soil_PH2	:=	INT_TO_REAL(MBdata_sensor_teplica_EC[4])/10;
			ELSE
				Modbus_array_errors[e_rs1]	:= sensor_teplica_EC_id;
				e_rs1	:= e_rs1+1;
			END_IF
			MB.ReadRegs(Execute:= FALSE);
			state:=15;

		END_IF

14:

		MB.ReadRegs(
			UnitID:= sensor_ponics_EC2_id,
			Quantity:= 1,
			MBAddr:= 8,
			cbLength:= 2,
			pMemoryAddr:= ADR(MBdata_sensor_ponics_EC2),
			Execute:= TRUE,
			Timeout:= timeoutvalue,
			Busy => busy,
		);
		IF NOT busy THEN
			IF (MB.Error = FALSE ) THEN
		(*	Modbus.Teplica_sensor_soil_Hum	:=	INT_TO_REAL(MBdata_sensor_teplica_EC[1])/10;
			Modbus.Teplica_sensor_soil_Temp	:=	INT_TO_REAL(MBdata_sensor_teplica_EC[2])/10;
			Modbus.Teplica_sensor_soil_PH2	:=	INT_TO_REAL(MBdata_sensor_teplica_EC[4])/10;
		*)
			ponics_EC2_1		:=	INT_TO_REAL(MBdata_sensor_ponics_EC2);
			Modbus.Sensor_EC2	:=	INT_TO_REAL(MBdata_sensor_ponics_EC2);
			ELSE
				Modbus_array_errors[e_rs1]	:= sensor_ponics_EC2_id;
				e_rs1	:= e_rs1+1;
			END_IF
			MB.ReadRegs(Execute:= FALSE);
			state:=15;

		END_IF





15:

		MB.ReadRegs(
			UnitID:= teplica_gate_pt1000_id,
			Quantity:= 8,
			MBAddr:= 32,
			cbLength:= 16,
			pMemoryAddr:= ADR(MBdata8_pt1000),
			Execute:= TRUE,
			Timeout:=  T#2000ms,
			Busy => busy,
		);
		IF NOT busy THEN
			IF (MB.Error = FALSE ) THEN
				IF (MBdata8_pt1000[1] <> -100)
					THEN	MBdata_teplica_gate_pt1000[1]:=INT_TO_REAL(MBdata8_pt1000[1])/10;
				END_IF
				IF (MBdata8_pt1000[2] <> -100)
					THEN	MBdata_teplica_gate_pt1000[2]:=INT_TO_REAL(MBdata8_pt1000[2])/10;
				END_IF
				IF (MBdata8_pt1000[3] <> -100)
					THEN	MBdata_teplica_gate_pt1000[3]:=INT_TO_REAL(MBdata8_pt1000[3])/10;
				END_IF
				IF (MBdata8_pt1000[4] <> -100)
					THEN	MBdata_teplica_gate_pt1000[4]:=INT_TO_REAL(MBdata8_pt1000[4])/10;
				END_IF
				IF (MBdata8_pt1000[5] <> -100)
					THEN	MBdata_teplica_gate_pt1000[5]:=INT_TO_REAL(MBdata8_pt1000[5])/10;
				END_IF
				IF (MBdata8_pt1000[6] <> -100)
					THEN	MBdata_teplica_gate_pt1000[6]:=INT_TO_REAL(MBdata8_pt1000[6])/10;
				END_IF
				IF (UINT_TO_INT(MBdata8_pt1000[7]) <> -100)
					THEN	MBdata_teplica_gate_pt1000[7]:=INT_TO_REAL(MBdata8_pt1000[7])/10;
				END_IF
				IF (MBdata8_pt1000[8] <> -100)
					THEN	MBdata_teplica_gate_pt1000[8]:=INT_TO_REAL(MBdata8_pt1000[8])/10;
				END_IF

				IF (MBdata_teplica_gate_pt1000[1] <> -100) THEN
					Modbus.Teplica_temp_LED	 	:=	MBdata_teplica_gate_pt1000[1];   (* Temp LED *)
				END_IF

				IF (MBdata_teplica_gate_pt1000[2] <> -100) THEN
					Modbus.Teplica_temp_panel		:= 	MBdata_teplica_gate_pt1000[2];  (* Temp panel*)
				END_IF

				IF (MBdata_teplica_gate_pt1000[3] <> -100) THEN
					Modbus.Teplica_temp_air_in	 	:=	MBdata_teplica_gate_pt1000[3];
				END_IF
				IF (MBdata_teplica_gate_pt1000[4] <> -100) THEN

					Modbus.Teplica_temp_ground		:=	MBdata_teplica_gate_pt1000[4];
				END_IF

				IF (MBdata_teplica_gate_pt1000[5] <> -100) THEN
					Modbus.Teplica_temp_water_tank 	:=	MBdata_teplica_gate_pt1000[5];
				END_IF

				IF (MBdata_teplica_gate_pt1000[6] <> -100) THEN
					Modbus.Teplica_temp_pipe_heat	:=	MBdata_teplica_gate_pt1000[6]; (* Temp air*)
				END_IF



			ELSE
				Modbus_array_errors[e_rs1]	:= teplica_gate_pt1000_id;
				e_rs1	:= e_rs1+1;
			END_IF
			MB.ReadRegs(Execute:= FALSE);
				state:=16;

		END_IF




16:

		MB.ReadRegs(
			UnitID:= Teplica_tank_level_id,
			Quantity:= 18,
			MBAddr:= 0,
			cbLength:= 36,
			pMemoryAddr:= ADR(teplica_tank_level_word),
			Execute:= TRUE,
			Timeout:= timeoutvalue,
			Busy => busy,
		);
		IF NOT busy THEN
			IF (mb.Error = FALSE ) THEN
				Teplica_tank_level		:=	WORD_TO_REAL(teplica_tank_level_word[4]);
				Modbus.Teplica_tank_level		:=	REAL_TO_INT(Teplica_tank_level);
(*				Modbus.Test5			:=	REAL_TO_INT(100*(Teplica_tank_level*0.001*3.14159*1.22*1.22*0.25)/1.5); *)
			ELSE
				Modbus_array_errors[e_rs1]	:= Teplica_tank_level_id;
				e_rs1	:= e_rs1+1;
			END_IF
			MB.ReadRegs(Execute:= FALSE);
			state:=17;
		END_IF

17:

		MB.ReadRegs(
			UnitID:= Teplica_tankA_level_id,
			Quantity:= 18, (* 1 *)
			MBAddr:= 0, (* 4 *)
			cbLength:= 36, (* 2 *)
			pMemoryAddr:= ADR(teplica_tankA_level_word),
			Execute:= TRUE,
			Timeout:= timeoutvalue,
			Busy => busy,
		);
		IF NOT busy THEN
			IF (mb.Error = FALSE ) THEN
				Teplica_tankA_level			:=	WORD_TO_REAL(teplica_tankA_level_word[4]);
				Modbus.Teplica_tankA_level	:=	REAL_TO_INT(Teplica_tankA_level)-8;
			ELSE
				Modbus_array_errors[e_rs1]	:= Teplica_tankA_level_id;
				e_rs1	:= e_rs1+1;
			END_IF
			MB.ReadRegs(Execute:= FALSE);
			state:=18;
		END_IF



18:

		MB.ReadRegs(
			UnitID:= Teplica_tankB_level_id,
			Quantity:= 18, (* 1 *)
			MBAddr:= 0, (* 4 *)
			cbLength:= 36, (* 2 *)
			pMemoryAddr:= ADR(teplica_tankB_level_word),
			Execute:= TRUE,
			Timeout:= timeoutvalue,
			Busy => busy,
		);
		IF NOT busy THEN
			IF (mb.Error = FALSE ) THEN
				Teplica_tankB_level			:=	WORD_TO_REAL(teplica_tankB_level_word[4]);
				Modbus.Teplica_tankB_level	:=	REAL_TO_INT(Teplica_tankB_level)-2;
			ELSE
				Modbus_array_errors[e_rs1]	:= Teplica_tankB_level_id;
				e_rs1	:= e_rs1+1;
			END_IF
			MB.ReadRegs(Execute:= FALSE);
			state:=20;
		END_IF


















20:

	IF (MBdataDO_byte <> MBdataDO_byte_read) THEN
		MB.WriteMultipleCoils(
			UnitID:= teplica_ADM4188_id,
			Quantity:= 8,
			MBAddr:= 0,
			cbLength:= 16,
			pMemoryAddr:= ADR(MBdataDO_byte),
			Execute:= TRUE,
			Timeout:= T#2000ms,
			Busy => busy,
			);
		IF NOT busy THEN
			IF (mb.Error = FALSE ) THEN
					cnt_clear_di_2	:=	TRUE;
			END_IF
			IF (mb.Error = TRUE ) THEN
				Modbus_array_errors[e_rs1]	:= teplica_ADM4188_id;
				e_rs1	:= e_rs1+1;
				cnt_clear_di_2	:=	FALSE;
			END_IF
			MB.ReadRegs(Execute:= FALSE);
			state:=21;
		END_IF
	ELSE
		state:=21;

	END_IF

(*считывание DO значений *)
21:
	MB.ReadCoils(
					UnitID:= teplica_ADM4188_id, (* station address *)
					Quantity:= 8,
					MBAddr:= 0,
					cbLength:= 16,
					pMemoryAddr:= ADR(MBdataDO_byte_read),
					Execute:= TRUE,
					Timeout:= T#2000ms,
					Busy => busy,
					);
		IF NOT busy THEN
			IF (mb.Error = FALSE ) THEN
					Teplica_DO1		:=MBdataDO_byte_read.0;
					Teplica_DO2		:=MBdataDO_byte_read.1;
					Teplica_DO3		:=MBdataDO_byte_read.2;
					Teplica_DO4		:=MBdataDO_byte_read.3;
					Teplica_DO5		:=MBdataDO_byte_read.4;
					Teplica_DO6		:=MBdataDO_byte_read.5;
					Teplica_DO7		:=MBdataDO_byte_read.6;
					Teplica_DO8		:=MBdataDO_byte_read.7;

			END_IF
(*			IF (mb.Error = TRUE ) THEN
				Modbus_array_errors[e_rs1]	:= teplica_ADM4188_id;
				e_rs1	:= e_rs1+1;
			END_IF
*)
			MB.ReadRegs(Execute:= FALSE);
			state:=105;
		END_IF



















(*	state:=105; *)

105: (*открываем канал*)


	Clear(Buffer := RxBufferCom1);
	arrSend[1]:=Merc_address;
	arrSend[2]:=1; (*код доступа*)
	arrSend[3]:=1; (*Уровень доступа*)

	MEMCPY(ADR(arrSend)+3,ADR(password_1),6); (*пароль*)
	crctest:=F_CRC16(ADR(arrSend),9); (*расчет контрольной суммы*)
	MEMCPY(ADR(arrSend)+9,ADR(crctest),SIZEOF(crctest)); (*прибавление контрольной суммы к запросу*)
	SendDatacom1(pSendData:=ADR(arrSend),Length:=11,TXBuffer:=TxBuffercom1,Busy=>,Error=>);
(*	tmCheck(in:=FALSE); *)
	tmCheckM(in:=FALSE);
	tmCheckM(in:=TRUE, pt:=t#3s); 	(*запуск таймера проверки - потеря связи\обрыв кабеля*)
	state:=106;

106: (*ответ*)
	ReceiveDatacom1(pPrefix:=,LenPrefix:=,pSuffix:=,LenSuffix:=,
	pReceiveData:=ADR(arrReceive),SizeReceiveData:=4,
	Timeout:=t#2s,Reset:=,
	RXbuffer:=RxBuffercom1,
	DataReceived=>,busy=>,Error=>,RxTimeout=>,LenReceiveData=>);
	IF ReceiveDatacom1.Error <> 0 THEN
		state:=888;
	END_IF
	IF receiveDatacom1.DataReceived THEN
		state:=107;
	ELSIF tmCheckM.Q THEN
		state:=888;
	END_IF
107: (*проверка ответа*)

	IF arrReceive[1] = Merc_address THEN
		state:= 108;
	ELSE
		state:=888;
	END_IF



108:
	(*	tmCheck(in:=FALSE);	*)
		tmCheck(in:=NOT tmCheck.q,pt:=t#2s);
		get_supply_done := FALSE;
		get_supply( byte1:=16#8, byte2:=16#16, byte3:=16#11,  supply1=>Modbus.UV1,supply2=>Modbus.UV2,supply3=>Modbus.UV3, done=>get_supply_done);
		IF get_supply_done = TRUE THEN
			Modbus.RS485_3_cnt_success := Modbus.RS485_3_cnt_success+1;
			state:=109;
		ELSIF tmcheck.Q THEN
			Modbus.RS485_3_cnt_error := Modbus.RS485_3_cnt_error+1;
			 state:=888;
		END_IF



 (*запрос на чтение тока  на всех фазах
--------------------------------------------------------------------------------------------------------------------------------------------------------------------
*)
109:
	(*	tmCheck(in:=FALSE);	*)
		tmCheck(in:=NOT tmCheck.q,pt:=t#2s);
		get_current_done := FALSE;
		get_current(byte1:=16#8, byte2:=16#16, byte3:=16#21,  current1=>Modbus.Ia1,current2=>Modbus.Ia2,current3=>Modbus.Ia3, done=>get_current_done);
		IF get_current_done = TRUE THEN
			state:=110;
		ELSIF tmcheck.Q THEN state:=888;
		END_IF

 (*запрос на чтение мощности  на всех фазах
--------------------------------------------------------------------------------------------------------------------------------------------------------------------
*)

110:
	(*	tmCheck(in:=FALSE);	*)
		tmCheck(in:=NOT tmCheck.q,pt:=t#2s);
		get_power_done := FALSE;
		get_power(byte1:=16#8, byte2:=16#16, byte3:=16#0,  power_total=>Modbus.pw_total, power1=>Modbus.pw1, power2=>Modbus.pw2,power3=>Modbus.pw3,done=>get_power_done);
		IF get_power_done = TRUE THEN
			state:=111;
		ELSIF tmcheck.Q THEN state:=888;
		END_IF

 (*запрос на чтение энергии T1
--------------------------------------------------------------------------------------------------------------------------------------------------------------------
*)
111:
	(*	tmCheck(in:=FALSE);	*)
		tmCheck(in:=NOT tmCheck.q,pt:=t#2s);
		get_energy_E_T1_done := FALSE;
		get_energy_E_T1(byte1:=5, byte2:=16#0, byte3:=1,  energy=>Modbus.E_T1, done=>get_energy_E_T1_done);
		IF get_energy_E_T1_done = TRUE THEN
			state:=112;
		ELSIF tmcheck.Q THEN state:=888;
		END_IF
 (*запрос на чтение энергии T2
--------------------------------------------------------------------------------------------------------------------------------------------------------------------
*)

112:
	(*	tmCheck(in:=FALSE);	*)
		tmCheck(in:=NOT tmCheck.q,pt:=t#2s);
		get_energy_E_T2_done := FALSE;
		get_energy_E_T2(byte1:=5, byte2:=16#0, byte3:=2,  energy=>Modbus.E_T2, done=>get_energy_E_T2_done);
		IF get_energy_E_T2_done = TRUE THEN
			state:=888;
		ELSIF tmcheck.Q THEN state:=888;
		END_IF

113:
		Timer_day(IN:=NOT Timer_dayQ , PT:=T#60m , Q=>Timer_dayQ , ET=> );
			IF timer_day.q THEN
				state:=114;
			ELSE
				state:=888;
			END_IF

114:
	(*	tmCheck(in:=FALSE);	*)
		tmCheckE(in:=NOT tmCheckE.q,pt:=t#2s, Q=>tmCheckEQ , ET=>);
		get_energy_MT_done := FALSE;

	(*	IF (tmCheckEQ) THEN *)
			get_energy_MT(byte1:=5, byte2:=INT_TO_BYTE(48+m), byte3:=INT_TO_BYTE(t),   energy=>energyMT[m,t],done=>get_energy_MT_done);
(*		END_IF *)

		IF get_energy_MT_done = TRUE THEN
			t:=t+1;
			IF (t>2 AND m<13) THEN
				t:=1;
				m:=m+1;
				state:=114;
			END_IF

					IF ( m=13) THEN
						t:=1;
						m:=1;
						Modbus.M1T1:=energyMT[1,1];
						Modbus.M1T2:=energyMT[1,2];
						Modbus.M2T1:=energyMT[2,1];
						Modbus.M2T2:=energyMT[2,2];
						Modbus.M3T1:=energyMT[3,1];
						Modbus.M3T2:=energyMT[3,2];
						Modbus.M4T1:=energyMT[4,1];
						Modbus.M4T2:=energyMT[4,2];
						Modbus.M5T1:=energyMT[5,1];
						Modbus.M5T2:=energyMT[5,2];
						Modbus.M6T1:=energyMT[6,1];
						Modbus.M6T2:=energyMT[6,2];
						Modbus.M7T1:=energyMT[7,1];
						Modbus.M7T2:=energyMT[7,2];
						Modbus.M8T1:=energyMT[8,1];
						Modbus.M8T2:=energyMT[8,2];
						Modbus.M9T1:=energyMT[9,1];
						Modbus.M9T2:=energyMT[9,2];
						Modbus.M10T1:=energyMT[10,1];
						Modbus.M10T2:=energyMT[10,2];
						Modbus.M11T1:=energyMT[11,1];
						Modbus.M11T2:=energyMT[11,2];
						Modbus.M12T1:=energyMT[12,1];
						Modbus.M12T2:=energyMT[12,2];
						state:=888;
					END_IF
		ELSIF tmcheckE.Q THEN state:=114;
		END_IF






888:
		Modbus_errors 				:=  BYTE_TO_DWORD(Modbus_array_errors[0]) + BYTE_TO_DWORD(Modbus_array_errors[1]) * 16#100 + BYTE_TO_DWORD(Modbus_array_errors[2]) * 16#10000 + BYTE_TO_DWORD(Modbus_array_errors[3]) * 16#1000000;
		Modbus.Modbus_4errors 		:= Modbus_errors;
		Modbus.Modbus_qual_errors	:= e_rs1;

		IF Modbus.Teplica_poliv_status_PLC=2 AND Modbus.Teplica_type_poliv = TRUE AND Poliv_liters>Modbus.Teplica_set_poliv_before_fert-10 AND MBdataDO_byte <> MBdataDO_byte_read THEN
			tTimerValue	:= t#1s;
		ELSE
			tTimerValue	:= t#60s;
		END_IF

		Timer1(IN:=NOT Timer1Q , PT:=tTimerValue , Q=>Timer1Q , ET=> );
		IF timer1.q THEN
			state:=0;
		END_IF

END_CASE

FtrigBusy(CLK:=mb.BUSY );
IF FtrigBusy.Q THEN
	IF mb.Error THEN
		LastModbusError := mb.ErrorDiagnostics;
		LastErrorstate := state;
		Modbus.RS485_1_cnt_error := Modbus.RS485_1_cnt_error + 1;
	ELSE
		Modbus.RS485_1_cnt_success := Modbus.RS485_1_cnt_success + 1;
	END_IF
END_IF



SerialLinecontrolCom1(
	mode:=SerialLinemode_kl6_22b_standard,
	pComIn:=ADR(RS485read.MB.InData),
	pComOut:=ADR(RS485read.MB.OutData),
	SizeComIn:=SIZEOF(RS485read.MB.OutData),
	TxBuffer:=TxBufferCom1,
	RxBuffer:=RxBufferCom1,
	Error=>,
	errorid=>);
END_PROGRAM

(* POU FB_GET_ENERGY, ST *)
FUNCTION_BLOCK FB_GET_ENERGY
VAR_INPUT
	byte1			: BYTE;
	byte2			: BYTE;
	byte3			: BYTE;
END_VAR

VAR_OUTPUT
	energy			: REAL;
	done			: BOOL;
END_VAR

VAR

	Clear				: ClearComBuffer;
	crctest				: WORD;
	arrReceive			: ARRAY[1..22] OF BYTE := 0,0,0,0,0,0,0,0,0,0,0,0,0,0,0,0,0,0,0,0,0,0;
	arrSend				: ARRAY[1..22] OF BYTE:= 0,0,0,0,0,0,0,0,0,0,0,0,0,0,0,0,0,0,0,0,0,0;
	state				: INT:= 0;
	dw_DATA			: DWORD:=0;
	E_active				: REAL:=0;
	E_reactive			: REAL:=0;
	tmcheck				: TON;
	CRC_calc			: WORD:=0;
	CRC_get				: WORD:=1;
END_VAR
tmcheck();

CASE state OF

0:
	done:=FALSE;
	Clear(Buffer := RxBufferCom1);
	arrSend[1]:=Merc_address;
	arrSend[2]:=byte1;
	arrSend[3]:=byte2;
	arrSend[4]:=byte3;

	crctest:=F_CRC16(ADR(arrSend), 4);
	MEMCPY(ADR(arrSend)+4,ADR(crctest),2);

	SendDataCom1(pSendData:=ADR(arrSend),length:=6,TXbuffer:=TXBufferCom1 );

	tmCheck(in:=FALSE);
	tmCheck(in:=TRUE,pt:=t#2s);
	state:=1;

1: (*ответ*)

	ReceiveDataCom1(pReceiveData:=ADR(arrReceive),SizeReceiveData:=19,TImeOut:=t#2s,Reset:=,RXbuffer:=RxBufferCom1);

	IF ReceiveDataCom1.Error <> 0 THEN
		state:=9;
	END_IF

	IF ReceiveDataCom1.DataReceived THEN
		state:=2;
	ELSIF tmcheck.Q THEN state:=9;
	END_IF;


2:(*расшифровка*)
	CRC_calc := F_CRC16(ADR(arrReceive), 17);
	MEMCPY(ADR(CRC_get),ADR(arrReceive[18]),1);
	MEMCPY(ADR(CRC_get)+1,ADR(arrReceive[19]),1);

	IF (  arrReceive[1] = Merc_address  AND CRC_calc = CRC_get ) THEN
			MEMCPY(ADR(dw_DATA),ADR(arrReceive[4]),2);
			MEMCPY(ADR(dw_DATA)+2,ADR(arrReceive[2]),2);
			E_active:=DWORD_TO_REAL(dw_DATA)/1000;(*активная мощ*)
			MEMCPY(ADR(dw_DATA),ADR(arrReceive[12]),2);
			MEMCPY(ADR(dw_DATA)+2,ADR(arrReceive[10]),2);
			E_reactive:=DWORD_TO_REAL(dw_DATA)/1000; (*реактивная мощность*)
			energy:=E_active;
			state:=10;
		ELSE state:=9;
	END_IF;
9:
	energy:=0;
	done := TRUE;
	state:=0;
10:
	done := TRUE;
	state:=0;

END_CASE;
END_FUNCTION_BLOCK

(* POU MB_func/F_CRC16, ST *)
FUNCTION F_CRC16 : WORD
VAR_INPUT
	pData: POINTER TO BYTE;		(* указатель на блок данных *)
	Size: WORD;						(* размер блока  данных *)
END_VAR
VAR
	Cnt: BYTE;							(* счетчик битов *)
END_VAR
F_CRC16 := 16#FFFF;
WHILE Size > 0 DO
	F_CRC16 := F_CRC16 XOR pData^;
	FOR Cnt := 0 TO 7 DO
		IF F_CRC16.0 = 0 THEN
			F_CRC16 := SHR(F_CRC16, 1);
		ELSE
			F_CRC16 := SHR(F_CRC16, 1) XOR 16#A001;
		END_IF
	END_FOR;
	pData := pData + 1;
	Size := Size - 1;
END_WHILE
END_FUNCTION

(* POU FB_GET_SUPPLY, ST *)
FUNCTION_BLOCK FB_GET_SUPPLY
VAR_INPUT
	byte1			: BYTE;
	byte2			: BYTE;
	byte3			: BYTE;

END_VAR

VAR_OUTPUT
	supply1			: REAL;
	supply2			: REAL;
	supply3			: REAL;
	done			: BOOL;
END_VAR

VAR

	Clear			: ClearComBuffer;
	crctest			: WORD;
	arrReceive		: ARRAY[1..12] OF BYTE := 0,0,0,0,0,0,0,0,0,0,0,0;
	arrSend			: ARRAY[1..6] OF BYTE:= 0,0,0,0,0,0;
	state			: INT:= 0;
	dw_DATA		: DWORD:=0;
	tmcheck			: TON;
	CRC_calc		: WORD:=0;
	CRC_get			: WORD:=1;

END_VAR
tmcheck();

CASE state OF

0:

	done:=FALSE;
	Clear(Buffer := RxBufferCom1);

	arrSend[1]:=Merc_address;
	arrSend[2]:=byte1;
	arrSend[3]:=byte2;
	arrSend[4]:=byte3;

	crctest:=F_CRC16(ADR(arrSend), 4);
	MEMCPY(ADR(arrSend)+4,ADR(crctest),2);

	SendDataCom1(pSendData:=ADR(arrSend),length:=6,TXbuffer:=TXBufferCom1 );

	tmCheck(in:=FALSE);
	tmCheck(in:=TRUE,pt:=t#2s);
	state:=1;

1: (*ответ*)

	ReceiveDataCom1(pReceiveData:=ADR(arrReceive),SizeReceiveData:=12,TImeOut:=t#2s,Reset:=,RXbuffer:=RxBufferCom1);

	IF ReceiveDataCom1.Error <> 0 THEN
		state:=9;
	END_IF

	IF ReceiveDataCom1.DataReceived THEN
		state:=2;

	ELSIF tmcheck.Q THEN state:=9;
	END_IF;


2:(*расшифровка*)
	(* arrReceive:=EchoDel(CheckUp:=TRUE, SentA:=arrSend, RecA:=arrReceive, Length:=UDINT_TO_INT(SendDataCom1.Length)); *)
	CRC_calc := F_CRC16(ADR(arrReceive), 10);
	MEMCPY(ADR(CRC_get),ADR(arrReceive[11]),1);
	MEMCPY(ADR(CRC_get)+1,ADR(arrReceive[12]),1);


	IF (  arrReceive[1] = Merc_address  AND CRC_calc = CRC_get ) THEN
		MEMCPY(ADR(dw_DATA),ADR(arrReceive[3]),1);
			MEMCPY(ADR(dw_DATA)+1,ADR(arrReceive[4]),1);
			arrReceive[2]:=arrReceive[2] AND 16#3F;
			MEMCPY(ADR(dw_DATA)+2,ADR(arrReceive[2]),1);
		supply1:=DWORD_TO_REAL(dw_DATA)/100;  (*Вольт*)

		MEMCPY(ADR(dw_DATA),ADR(arrReceive[6]),1);
			MEMCPY(ADR(dw_DATA)+1,ADR(arrReceive[7]),1);
			arrReceive[5]:=arrReceive[5] AND 16#3F;
			MEMCPY(ADR(dw_DATA)+2,ADR(arrReceive[5]),1);
		supply2:=DWORD_TO_REAL(dw_DATA)/100;  (*Вольт*)

		MEMCPY(ADR(dw_DATA),ADR(arrReceive[9]),1);
			MEMCPY(ADR(dw_DATA)+1,ADR(arrReceive[10]),1);
			arrReceive[8]:=arrReceive[8] AND 16#3F;
			MEMCPY(ADR(dw_DATA)+2,ADR(arrReceive[8]),1);
		supply3:=DWORD_TO_REAL(dw_DATA)/100;  (*Вольт*)



			state:=10;
		ELSE state:=9;
	END_IF;

9:
	supply1:=0;
	supply2:=0;
	supply3:=0;
	done := TRUE;
	state:=0;

10:
	done := TRUE;
	state:=0;

END_CASE;
END_FUNCTION_BLOCK

(* POU FB_GET_CURRENT, ST *)
FUNCTION_BLOCK FB_GET_CURRENT
VAR_INPUT
	byte1			: BYTE;
	byte2			: BYTE;
	byte3			: BYTE;

END_VAR

VAR_OUTPUT
	current1			: REAL;
	current2			: REAL;
	current3			: REAL;
	done			: BOOL;
END_VAR

VAR
	Clear			: ClearComBuffer;
	crctest			: WORD;
	arrReceive		: ARRAY[1..12] OF BYTE := 0,0,0,0,0,0,0,0,0,0,0,0;
	arrSend			: ARRAY[1..6] OF BYTE:= 0,0,0,0,0,0;
	state			: INT:= 0;
	dw_DATA		: DWORD:=0;
	tmcheck			: TON;
	CRC_calc		: WORD:=0;
	CRC_get			: WORD:=1;
END_VAR
tmcheck();

CASE state OF

0:
	done:=FALSE;
	Clear(Buffer := RxBufferCom1);
	arrSend[1]:=Merc_address;
	arrSend[2]:=byte1;
	arrSend[3]:=byte2;
	arrSend[4]:=byte3;

	crctest:=F_CRC16(ADR(arrSend), 4);
	MEMCPY(ADR(arrSend)+4,ADR(crctest),2);

	SendDataCom1(pSendData:=ADR(arrSend),length:=6,TXbuffer:=TXBufferCom1 );

	tmCheck(in:=FALSE);
	tmCheck(in:=TRUE,pt:=t#2s);
	state:=1;

1: (*ответ*)

	ReceiveDataCom1(pReceiveData:=ADR(arrReceive),SizeReceiveData:=12,TImeOut:=t#2s,Reset:=,RXbuffer:=RxBufferCom1);

	IF ReceiveDataCom1.Error <> 0 THEN
		state:=9;
	END_IF

	IF ReceiveDatacom1.DataReceived THEN
		state:=2;
	ELSIF tmcheck.Q THEN state:=9;
	END_IF;


2:(*расшифровка*)

	CRC_calc := F_CRC16(ADR(arrReceive), 10);
	MEMCPY(ADR(CRC_get),ADR(arrReceive[11]),1);
	MEMCPY(ADR(CRC_get)+1,ADR(arrReceive[12]),1);


	IF (  arrReceive[1] = Merc_address  AND CRC_calc = CRC_get ) THEN

			MEMCPY(ADR(dw_DATA),ADR(arrReceive[3]),1);
			MEMCPY(ADR(dw_DATA)+1,ADR(arrReceive[4]),1);
			arrReceive[2]:=arrReceive[2] AND 16#3F;
			MEMCPY(ADR(dw_DATA)+2,ADR(arrReceive[2]),1);
			current1 :=DWORD_TO_REAL(dw_DATA)/1000;  (*Ампер*)

			MEMCPY(ADR(dw_DATA),ADR(arrReceive[6]),1);
			MEMCPY(ADR(dw_DATA)+1,ADR(arrReceive[7]),1);
			arrReceive[5]:=arrReceive[5] AND 16#3F;
			MEMCPY(ADR(dw_DATA)+2,ADR(arrReceive[5]),1);
			current2:=DWORD_TO_REAL(dw_DATA)/1000;  (*Ампер*)

			MEMCPY(ADR(dw_DATA),ADR(arrReceive[9]),1);
			MEMCPY(ADR(dw_DATA)+1,ADR(arrReceive[10]),1);
			arrReceive[8]:=arrReceive[8] AND 16#3F;
			MEMCPY(ADR(dw_DATA)+2,ADR(arrReceive[8]),1);
			current3 :=DWORD_TO_REAL(dw_DATA)/1000;  (*Ампер*)
			state:=10;
		ELSE state:=9;
	END_IF;

9:
	current1:=0;
	current2:=0;
	current3:=0;
	done := TRUE;
	state:=0;
10:
	done := TRUE;
	state:=0;

END_CASE;
END_FUNCTION_BLOCK

(* POU FB_GET_POWER, ST *)
FUNCTION_BLOCK FB_GET_POWER
VAR_INPUT
	byte1			: BYTE;
	byte2			: BYTE;
	byte3			: BYTE;
END_VAR

VAR_OUTPUT
	power_total		: REAL;
	power1			: REAL;
	power2			: REAL;
	power3			: REAL;
	done			: BOOL;
END_VAR

VAR
	Clear				: ClearComBuffer;
	crctest				: WORD;
	arrReceive			: ARRAY[1..15] OF BYTE := 0,0,0,0,0,0,0,0,0,0,0,0,0,0,0;
	arrSend				: ARRAY[1..6] OF BYTE:= 0,0,0,0,0,0;
	state				: INT:= 0;
	dw_DATA			: DWORD:=0;
	tmcheck				: TON;
	CRC_calc			: WORD:=0;
	CRC_get				: WORD:=1;
END_VAR
tmcheck();

CASE state OF

0:
	done:=FALSE;
	Clear(Buffer := RxBufferCom1);
	arrSend[1]:=Merc_address;
	arrSend[2]:=byte1;
	arrSend[3]:=byte2;
	arrSend[4]:=byte3;

	crctest:=F_CRC16(ADR(arrSend), 4);
	MEMCPY(ADR(arrSend)+4,ADR(crctest),2);

	SendDataCom1(pSendData:=ADR(arrSend),length:=6,TXbuffer:=TXBufferCom1 );

	tmCheck(in:=FALSE);
	tmCheck(in:=TRUE,pt:=t#2s);
	state:=1;

1: (*ответ*)

	ReceiveDataCom1(pReceiveData:=ADR(arrReceive),SizeReceiveData:=15,TImeOut:=t#2s,Reset:=,RXbuffer:=RxBufferCom1);

	IF ReceiveDataCom1.Error <> 0 THEN
		state:=9;
	END_IF

	IF ReceiveDataCom1.DataReceived THEN
		state:=2;
	ELSIF tmcheck.Q THEN state:=9;
	END_IF;


2:(*расшифровка*)
	CRC_calc := F_CRC16(ADR(arrReceive), 13);
	MEMCPY(ADR(CRC_get),ADR(arrReceive[14]),1);
	MEMCPY(ADR(CRC_get)+1,ADR(arrReceive[15]),1);


	IF (  arrReceive[1] = Merc_address  AND CRC_calc = CRC_get ) THEN
			MEMCPY(ADR(dw_DATA),ADR(arrReceive[3]),1);
			MEMCPY(ADR(dw_DATA)+1,ADR(arrReceive[4]),1);
			arrReceive[2]:=arrReceive[2] AND 16#3F;
			MEMCPY(ADR(dw_DATA)+2,ADR(arrReceive[2]),1);
			power_total:=DWORD_TO_REAL(dw_DATA)/100;

			MEMCPY(ADR(dw_DATA),ADR(arrReceive[6]),1);
			MEMCPY(ADR(dw_DATA)+1,ADR(arrReceive[7]),1);
			arrReceive[5]:=arrReceive[5] AND 16#3F;
			MEMCPY(ADR(dw_DATA)+2,ADR(arrReceive[5]),1);
			power1:=DWORD_TO_REAL(dw_DATA)/100;

			MEMCPY(ADR(dw_DATA),ADR(arrReceive[9]),1);
			MEMCPY(ADR(dw_DATA)+1,ADR(arrReceive[10]),1);
			arrReceive[8]:=arrReceive[8] AND 16#3F;
			MEMCPY(ADR(dw_DATA)+2,ADR(arrReceive[8]),1);
			power2:=DWORD_TO_REAL(dw_DATA)/100;

			MEMCPY(ADR(dw_DATA),ADR(arrReceive[12]),1);
			MEMCPY(ADR(dw_DATA)+1,ADR(arrReceive[13]),1);
			arrReceive[11]:=arrReceive[11] AND 16#3F;
			MEMCPY(ADR(dw_DATA)+2,ADR(arrReceive[11]),1);
			power3:=DWORD_TO_REAL(dw_DATA)/100;



			state:=10;
		ELSE state:=9;
	END_IF;

9:
	power_total:=0;
	power1:=0;
	power2:=0;
	power3:=0;

	done := TRUE;
	state:=0;
10:
	done := TRUE;
	state:=0;

END_CASE;
END_FUNCTION_BLOCK

(* POU RS485read_2, ST *)
PROGRAM RS485read_2
VAR

(*	KLConfiguration: KL6configuration; *)
(*	Period_vent_switch	: INT:=180; *)
	tTimerValue			: TIME	:=	t#60s; (* Период опроса RS485*)

	MBdata_pzem			 : ARRAY [1..2] OF INT;

	FtrigBusy				: F_TRIG;
	timeoutvalue				: TIME := T#2000ms;		(* timeout while waiting for an answer of the modbus slave *)
	state					: INT;
	busy					: BOOL;
	LastErrorstate				: INT;
	LastModbusError			: ST_ModbusErrorDiagnostics;
	CounterError				: DINT;
	CounterSuccess			: DINT;

	sensors_PZEM_id			: BYTE:=16#02;
	sensors_PZEM_data		: ARRAY[1..2] OF REAL:=2(0);

(*	sensors_DS18B20_id			: BYTE:=16#01;
	sensors_DS18B20_temp		: ARRAY[1..8] OF REAL:=8(0);
*)
(*
	get_co2_mh_z19b_1floor	: FB_GET_CO2_MH_Z19B;
	get_co2_mh_z19b_1floor_done	: BOOL;
*)




	PWM_YC110_id			: BYTE:= 16#20 ; (*32 *)
	PWM_levels				 : ARRAY [1..4] OF INT;	(* reg dec 32*)
	PWM_levels_mem		 : ARRAY [1..4] OF INT;
	PWM_freq				 : ARRAY [1..4] OF INT; (* reg dec 64*)
	PWM_freq_mem			 : ARRAY [1..4] OF INT;
	PWM_cycle				 : ARRAY [1..4] OF INT;

	PWM_param_polar		:  INT;	(* reg dec 18*)
	PWM_param_polar_1		:  INT:=1;
	PWM_param_prz			: INT;	(* reg dec 30*)
	PWM_param_prz_1		: INT:=1;	(* reg dec 30*)

	PWM_cycle_1			:  UINT:=65535;
	PWM_cycle_2			:  UINT:=65535;
	PWM_cycle_3			:  UINT:=65535;
	PWM_cycle_4			:  UINT:=65535;

	PWM_set_freq			: INT:=300;
	set_param				: BOOL;
END_VAR
(*Modbus.RS485_2_cnt_error		:= CounterError;
Modbus.RS485_2_cnt_success	:= Modbus.RS485_2_cnt_success; *)




CASE state OF
0:
		MB2.ReadRegs(Execute:= FALSE);
		state := 1;

1:

		MB2.ReadInputRegs(
			UnitID:= sensors_PZEM_id,
			Quantity:= 2,
			MBAddr:= 0,
			cbLength:= 4,
			pMemoryAddr:= ADR(MBdata_pzem),
			Execute:= TRUE,
			Timeout:= timeoutvalue,
			Busy => busy,
		);
		IF NOT busy THEN
			IF (mb2.Error = FALSE ) THEN
				sensors_PZEM_data[1]:=INT_TO_REAL(MBdata_pzem[1])/100;
				sensors_PZEM_data[2]:=INT_TO_REAL(MBdata_pzem[2])/100;
				Modbus.DC_Uv:=sensors_PZEM_data[1];
				Modbus.DC_Ia:=sensors_PZEM_data[2];

			END_IF
			MB2.ReadRegs(Execute:= FALSE);
			state:=888;

		END_IF



2:
	MB2.WriteSingleRegister(
					UnitID:= PWM_YC110_id, (* station address *)
					Quantity:= 1,
					MBAddr:= 32,
					cbLength:= 2,
					pMemoryAddr:= ADR(fert_pwm_levelA),
					Execute:= TRUE,
					Timeout:= T#1000ms,
					Busy => busy,
					);
		IF NOT busy THEN
		(*	IF (MB2.Error = FALSE ) THEN

			END_IF
		*)
			MB2.ReadRegs(Execute:= FALSE);
			state:=3;
		END_IF

3:
	MB2.WriteSingleRegister(
					UnitID:= PWM_YC110_id, (* station address *)
					Quantity:= 1,
					MBAddr:= 33,
					cbLength:= 2,
					pMemoryAddr:= ADR(fert_pwm_levelB),
					Execute:= TRUE,
					Timeout:= T#1000ms,
					Busy => busy,
					);
		IF NOT busy THEN
		(*	IF (MB2.Error = FALSE ) THEN

			END_IF
		*)
			MB2.ReadRegs(Execute:= FALSE);
			state:=4;
		END_IF






4:
IF (set_param= FALSE) THEN
	MB2.WriteSingleRegister(
					UnitID:= PWM_YC110_id, (* station address *)
					Quantity:= 1,
					MBAddr:= 30,
					cbLength:= 2,
					pMemoryAddr:=ADR(PWM_param_prz_1) ,
					Execute:= TRUE,
					Timeout:= T#1000ms,
					Busy => busy,
					);
		IF NOT busy THEN
			MB2.ReadRegs(Execute:= FALSE);
			state:=5;
		END_IF
ELSE
	state:=11;
END_IF





5:
	MB2.WriteSingleRegister(
					UnitID:= PWM_YC110_id, (* station address *)
					Quantity:= 1,
					MBAddr:= 96,
					cbLength:= 2,
					pMemoryAddr:=ADR(PWM_cycle_1) ,
					Execute:= TRUE,
					Timeout:= T#1000ms,
					Busy => busy,
					);
		IF NOT busy THEN
		(*	IF (MB2.Error = FALSE ) THEN

			END_IF
		*)
			MB2.ReadRegs(Execute:= FALSE);
			state:=7;
		END_IF


7:
	MB2.WriteSingleRegister(
					UnitID:= PWM_YC110_id, (* station address *)
					Quantity:= 1,
					MBAddr:= 97,
					cbLength:= 2,
					pMemoryAddr:=ADR(PWM_cycle_2) ,
					Execute:= TRUE,
					Timeout:= T#1000ms,
					Busy => busy,
					);
		IF NOT busy THEN
		(*	IF (MB2.Error = FALSE ) THEN

			END_IF
		*)
			MB2.ReadRegs(Execute:= FALSE);
			state:=8;
		END_IF


8:
	MB2.WriteSingleRegister(
					UnitID:= PWM_YC110_id, (* station address *)
					Quantity:= 1,
					MBAddr:= 98,
					cbLength:= 2,
					pMemoryAddr:=ADR(PWM_cycle_3) ,
					Execute:= TRUE,
					Timeout:= T#1000ms,
					Busy => busy,
					);
		IF NOT busy THEN
		(*	IF (MB2.Error = FALSE ) THEN

			END_IF
		*)
			MB2.ReadRegs(Execute:= FALSE);
			state:=9;
		END_IF

9:
	MB2.WriteSingleRegister(
					UnitID:= PWM_YC110_id, (* station address *)
					Quantity:= 1,
					MBAddr:= 99,
					cbLength:= 2,
					pMemoryAddr:=ADR(PWM_cycle_4) ,
					Execute:= TRUE,
					Timeout:= T#1000ms,
					Busy => busy,
					);
		IF NOT busy THEN
		(*	IF (MB2.Error = FALSE ) THEN

			END_IF
		*)
			MB2.ReadRegs(Execute:= FALSE);
			state:=10;
		END_IF




10:
	MB2.WriteSingleRegister(
					UnitID:= PWM_YC110_id, (* station address *)
					Quantity:= 1,
					MBAddr:= 64,
					cbLength:= 2,
					pMemoryAddr:=ADR(PWM_set_freq) ,
					Execute:= TRUE,
					Timeout:= T#1000ms,
					Busy => busy,
					);
		IF NOT busy THEN
		(*	IF (MB2.Error = FALSE ) THEN

			END_IF
		*)
			MB2.ReadRegs(Execute:= FALSE);
			set_param:= TRUE;
			state:=11;
		END_IF







11:
	MB2.ReadRegs(
					UnitID:= PWM_YC110_id, (* station address *)
					Quantity:= 1,
					MBAddr:= 18,
					cbLength:= 2,
					pMemoryAddr:= ADR(PWM_param_polar),
					Execute:= TRUE,
					Timeout:= T#1000ms,
					Busy => busy,
					);
		IF NOT busy THEN
		(*	IF (MB2.Error = FALSE ) THEN

			END_IF
		*)
			MB2.ReadRegs(Execute:= FALSE);
			state:=12;
		END_IF

12:
	MB2.ReadRegs(
					UnitID:= PWM_YC110_id, (* station address *)
					Quantity:= 4,
					MBAddr:= 96,
					cbLength:= 8,
					pMemoryAddr:= ADR(PWM_cycle),
					Execute:= TRUE,
					Timeout:= T#1000ms,
					Busy => busy,
					);
		IF NOT busy THEN
		(*	IF (MB2.Error = FALSE ) THEN

			END_IF
		*)
			MB2.ReadRegs(Execute:= FALSE);
			state:=13;
		END_IF



13:
	MB2.ReadRegs(
					UnitID:= PWM_YC110_id, (* station address *)
					Quantity:= 4,
					MBAddr:= 32,
					cbLength:= 8,
					pMemoryAddr:= ADR(PWM_levels),
					Execute:= TRUE,
					Timeout:= T#1000ms,
					Busy => busy,
					);
		IF NOT busy THEN
			IF (MB2.Error = FALSE ) THEN
				PWM_levels_mem[1]	:=	PWM_levels[1];
				PWM_levels_mem[2]	:=	PWM_levels[2];
				PWM_levels_mem[3]	:=	PWM_levels[3];
				PWM_levels_mem[4]	:=	PWM_levels[4];

			END_IF

			MB2.ReadRegs(Execute:= FALSE);
			state:=14;
		END_IF

14:
	MB2.ReadRegs(
					UnitID:= PWM_YC110_id, (* station address *)
					Quantity:= 4,
					MBAddr:= 64,
					cbLength:= 8,
					pMemoryAddr:= ADR(PWM_freq),
					Execute:= TRUE,
					Timeout:= T#1000ms,
					Busy => busy,
					);
		IF NOT busy THEN
			IF (MB2.Error = FALSE ) THEN
				PWM_freq_mem[1]	:=	PWM_freq[1];
				PWM_freq_mem[2]	:=	PWM_freq[2];
				PWM_freq_mem[3]	:=	PWM_freq[3];
				PWM_freq_mem[4]	:=	PWM_freq[4];

			END_IF

			MB2.ReadRegs(Execute:= FALSE);
			state:=888;
		END_IF

(*

5:
	MB2.ReadRegs(
					UnitID:= PWM_YC110_id, (* station address *)
					Quantity:= 1,
					MBAddr:= 30,
					cbLength:= 2,
					pMemoryAddr:= ADR(PWM_param_prz),
					Execute:= TRUE,
					Timeout:= T#1000ms,
					Busy => busy,
					);
		IF NOT busy THEN
		(*	IF (MB2.Error = FALSE ) THEN

			END_IF
		*)
			MB2.ReadRegs(Execute:= FALSE);
			state:=6;
		END_IF

*)


888:
		TimerRS485_2(IN:=NOT TimerRS485_2Q , PT:=tTimerValue , Q=>TimerRS485_2Q , ET=> );
		IF TimerRS485_2.q THEN
			state:=0;
		END_IF

END_CASE

FtrigBusy(CLK:=mb2.BUSY );
IF FtrigBusy.Q THEN
	IF mb2.Error THEN
		LastModbusError := mb2.ErrorDiagnostics;
		LastErrorstate := state;
		Modbus.RS485_2_cnt_error := Modbus.RS485_2_cnt_error + 1;
	ELSE
		Modbus.RS485_2_cnt_success := Modbus.RS485_2_cnt_success + 1;
	END_IF
END_IF

SerialLinecontrolCom2(
	mode:=SerialLinemode_kl6_5b_standard,
	pComIn:=ADR(RS485read_2.MB2.InData),
	pComOut:=ADR(RS485read_2.MB2.OutData),
	SizeComIn:=SIZEOF(RS485read_2.MB2.OutData),
	TxBuffer:=TxBufferCom2,
	RxBuffer:=RxBufferCom2,
	Error=>,
	errorid=>);
END_PROGRAM

(* POU VentControl, ST *)
PROGRAM VentControl
VAR
	Temperature_max_to_heat	: REAL:=17;		(* Максимальная температура наружнего воздуха при которой разрешено включать воздухонагреватель*)
	gisterezis				: REAL:=0.2;	(* Гистерезис  разрешения включения воздухонагревателя, градусы цельсия *)
	vent_valve_opened	 	: BOOL:=FALSE;	(*После перезагрузки ПЛК считаем что приточный клапан закрыт *)
	Period_start_delay		: INT:=60; 	(* Время задержки включения вентилятора после сигнала на открытие приточного клапана, сек *)
	Period_stop_delay		: INT:=60;		(* Время задержки отключения вентилятора после сигнала на останов вентиляции - для остужения разогретых ТЭНов воздухонагревателя, сек *)
	Timer1					: TON;		(* Таймер задержки включения вентилятора после сигнала на открытие приточного клапана *)
	Timer2					: TON;		(* Таймер задержки отключения вентилятора после сигнала на останов вентиляции - для остужения разогретых ТЭНов воздухонагревателя *)
	Timer1Q					: BOOL;
	Timer2Q					: BOOL;
	tTimerValue1				: TIME;
	tTimerValue2				: TIME;
END_VAR
tTimerValue1 := DINT_TO_TIME(Period_start_delay*1000);
tTimerValue2 := DINT_TO_TIME(Period_stop_delay*1000);

IF (Modbus.Vent=FALSE) THEN
	HW_vent_in_heat := FALSE;
	vent_valve_opened := FALSE;
	HW_vent_valve_input:=FALSE;
	Timer2(IN:=NOT Timer2Q , PT:=tTimerValue2 , Q=>Timer2Q , ET=> );
	IF timer2q THEN
		HW_trans_power:=FALSE;
	END_IF


ELSE
	HW_vent_valve_input:=TRUE;
(*	HW_vent_valve_output:=TRUE; *)

	IF (vent_valve_opened = FALSE) THEN
		Timer1(IN:=NOT Timer1Q , PT:=tTimerValue1 , Q=>Timer1Q , ET=> );
		IF timer1.q THEN
			vent_valve_opened := TRUE;
		END_IF
	END_IF

	IF (vent_valve_opened=TRUE) THEN
		HW_trans_power:=TRUE;
		IF (HW_vent_relay_pressure=TRUE) THEN
			IF (Modbus.Vent_heat=2) THEN
				IF (Modbus.Street_temp < Temperature_max_to_heat-gisterezis) THEN
					HW_vent_in_heat:=TRUE;
				END_IF
				IF (Modbus.Street_temp > Temperature_max_to_heat+gisterezis) THEN
					HW_vent_in_heat:=FALSE;
				END_IF
			ELSE
				IF (Modbus.Vent_heat=1) THEN
					HW_vent_in_heat:=TRUE;
				END_IF
				IF (Modbus.Vent_heat=0) THEN
					HW_vent_in_heat:=FALSE;
				END_IF
			END_IF
		END_IF   (*vent_relay_pressure*)
	END_IF (*vent_valve_opened*)
END_IF (*Vent*)
END_PROGRAM

(* POU VentPower, ST *)
PROGRAM VentPower
VAR
	Vent_power			: REAL:=30;  (* После перезагрузки ПЛК задаём начальную мощность условных 30%  *)
	CO2_old				: REAL:=410; (* После перезагрузки ПЛК задаём принудительно последнее значение CO2 = 410 (абсолютно свежий воздух) *)
	Period_vent_switch	: INT:=180; (* Частота переключения режимов работы вентилятора по показаниям датчиков CO2, секунды*)
	Timer1				: TON;
	Timer1Q				: BOOL;
	count				: INT:=0;
	CO2_max			: REAL;
	tTimerValue			: TIME;

END_VAR
tTimerValue := DINT_TO_TIME(Period_vent_switch*1000);

IF (Modbus.Vent =TRUE  ) THEN

	Timer1(IN:=NOT Timer1Q , PT:=tTimerValue , Q=>Timer1Q , ET=> );

	IF timer1.q THEN
	CO2_max:=MAX (Modbus.First_floor_CO2, Modbus.Second_floor_CO2);

	IF (  (CO2_max >=  CO2_old-10 )  AND ( CO2_max >  INT_TO_REAL(Modbus.Target_CO2)*1.05 ) ) THEN
			Vent_power:=Vent_power+5;
		END_IF
		count:=count+1;

		IF (count = 2)	THEN
			IF (  CO2_max <=  INT_TO_REAL(Modbus.Target_CO2)*0.99) THEN
				Vent_power:=Vent_power-1;
			END_IF
		count:=1;
		END_IF

		IF (Vent_power>80) THEN
			Vent_power:=80;
		END_IF
		IF(Vent_power<20) THEN
			Vent_power:=20;
		END_IF

		IF (Vent_Power > 75 AND Modbus.Street_temp > -10  ) THEN

					Modbus.Vent_input_level:=200;	(*200 м. куб в час при подаче напряжения на вентилятор  220V *)
					HW_vent_in_trans_160_220:=FALSE;
					HW_vent_in_trans_LO_HI:=FALSE;

			ELSIF (Vent_Power>50 AND Modbus.Street_temp > -14) THEN
					Modbus.Vent_input_level:=180; (*200 м. куб в час при подаче напряжения на вентилятор 220V *)
					HW_vent_in_trans_160_220:=FALSE;
					HW_vent_in_trans_LO_HI:=FALSE;

			ELSIF (Vent_Power>35  AND Modbus.Street_temp > -20) THEN

					Modbus.Vent_input_level:=150; (* 150 м. куб в час при подаче напряжения на вентилятор160V *)
					HW_vent_in_trans_160_220:=TRUE;
					HW_vent_in_trans_LO_HI:=FALSE;


			ELSIF (Vent_Power>25 ) THEN

					Modbus.Vent_input_level:=110; (* 110 м. куб в час при подаче напряжения на вентилятор 130V *)
					HW_vent_in_trans_105_130:=FALSE;
					HW_vent_in_trans_LO_HI:=TRUE;


			ELSE
				Modbus.Vent_input_level:=80; (* 80 м. куб в час при подаче напряжения на вентилятор 105V *)
				HW_vent_in_trans_105_130:=TRUE;
				HW_vent_in_trans_LO_HI:=TRUE;


			END_IF

			CO2_old:=CO2_max;

		END_IF	(* Timer1 *)

	ELSE	 (* Vent=TRUE*)


		Modbus.Vent_input_level:=0;

END_IF   (* Vent=TRUE*)
END_PROGRAM

(* POU Poliv, ST *)
PROGRAM Poliv
VAR
	TRIG_poliv_terrasa	:	R_TRIG;
	TRIG_poliv_zapad	:	R_TRIG;
	TRIG_poliv_south		:	R_TRIG;
	TRIG_poliv_north		:	R_TRIG;
	TRIG_poliv_flowers		:	R_TRIG;

	Period_pomp_garden_delay	: INT:=15;				(* Задержка включения насоса после сигнала на открытие клапана=15 сек. *)

 	 tTimerValue_zapad			: TIME;
	Timer_poliv_zapad			: TON;
	Timer_poliv_zapadQ			:  BOOL;
	 tTimerValue_zapad_est		: TIME;

	tTimerValue_terrasa			: TIME;
	Timer_poliv_terrasa			: TON;
	Timer_poliv_terrasaQ			:  BOOL;
	tTimerValue_terrasa_est		: TIME;

	 tTimerValue_south			: TIME;
	Timer_poliv_south				: TON;
	Timer_poliv_southQ			:  BOOL;
	 tTimerValue_south_est		: TIME;


 	tTimerValue_north				: TIME;
	Timer_poliv_north				: TON;
	Timer_poliv_northQ			:  BOOL;
 	tTimerValue_north_est			: TIME;


 	tTimerValue_flowers				: TIME;
	Timer_poliv_flowers				: TON;
	Timer_poliv_flowersQ			:  BOOL;
 	tTimerValue_flowers_est			: TIME;


	TON_pomp_garden			: TON ;
	pomp_garden_start			: BOOL;

	tTimerValue					: TIME;
END_VAR
tTimerValue := DINT_TO_TIME(Period_pomp_garden_delay*1000);


Timer_poliv_zapad();
Timer_poliv_terrasa();
Timer_poliv_south();
Timer_poliv_north();
Timer_poliv_flowers();

IF (Modbus.Poliv_valve_winter = FALSE) THEN


	TRIG_poliv_terrasa(CLK :=HW_button_poliv_terrasa);
	TRIG_poliv_zapad(CLK :=HW_button_poliv_zapad);
	TRIG_poliv_south(CLK :=HW_button_poliv_south);
	TRIG_poliv_north(CLK :=HW_button_poliv_north);





	IF (TRIG_poliv_terrasa.Q) THEN
		IF (Modbus.Poliv_terrasa = TRUE ) THEN
			Modbus.Poliv_terrasa := FALSE;
		ELSE
			Modbus.Poliv_terrasa := TRUE;
			Modbus.Poliv_terrasa_minutes:=120;
		END_IF

	END_IF



	IF (TRIG_poliv_zapad.Q) THEN
		IF (Modbus.Poliv_zapad = TRUE ) THEN
			Modbus.Poliv_zapad := FALSE;
		ELSE
			Modbus.Poliv_zapad := TRUE;
			Modbus.Poliv_zapad_minutes:=120;
		END_IF

	END_IF


	IF (TRIG_poliv_south.Q) THEN
		IF (Modbus.Poliv_south = TRUE ) THEN
			Modbus.Poliv_south := FALSE;
		ELSE
			Modbus.Poliv_south_minutes:=120;
			Modbus.Poliv_south := TRUE;
		END_IF

	END_IF


	IF (TRIG_poliv_north.Q) THEN
		IF (Modbus.Poliv_north = TRUE ) THEN
			Modbus.Poliv_north := FALSE;
		ELSE
			Modbus.Poliv_north_minutes:=120;
			Modbus.Poliv_north := TRUE;
		END_IF

	END_IF


	Modbus.Poliv_zapad_minutes_est	:= TIME_TO_INT(Timer_poliv_zapad.ET/(60*1000));
	Modbus.Poliv_terrasa_minutes_est	:=  TIME_TO_INT(Timer_poliv_terrasa.ET/(60*1000));
	Modbus.Poliv_south_minutes_est	:=  TIME_TO_INT(Timer_poliv_south.ET/(60*1000));
	Modbus.Poliv_north_minutes_est	:=  TIME_TO_INT(Timer_poliv_north.ET/(60*1000));
	Modbus.Poliv_flowers_minutes_est	:=  TIME_TO_INT(Timer_poliv_flowers.ET/(60*1000));


	IF (Modbus.Poliv_zapad = TRUE ) THEN
		tTimerValue_zapad := DINT_TO_TIME(Modbus.Poliv_zapad_minutes*60*1000);
		HW_poliv_zapad	:=	TRUE;
		Timer_poliv_zapad(IN:=NOT Timer_poliv_zapadQ , PT:=tTimerValue_zapad , Q=>Timer_poliv_zapadQ , ET=>tTimerValue_zapad_est );

	END_IF
	IF (Modbus.Poliv_zapad = FALSE ) THEN
		HW_poliv_zapad	:=	FALSE;
		Timer_poliv_zapadQ := FALSE;
		Timer_poliv_zapad(IN:=FALSE , PT:=T#0ms , Q=>Timer_poliv_zapadQ , ET=>tTimerValue_zapad_est );
	END_IF
	IF Timer_poliv_zapad.q THEN
		Modbus.Poliv_zapad := FALSE;
		HW_poliv_zapad	:=	FALSE;
	END_IF
	
	
	
	
	IF (Modbus.Poliv_terrasa = TRUE ) THEN
		tTimerValue_terrasa := DINT_TO_TIME(Modbus.Poliv_terrasa_minutes*60*1000);
		HW_poliv_terrasa	:=	TRUE;
		Timer_poliv_terrasa(IN:=NOT Timer_poliv_terrasaQ , PT:=tTimerValue_terrasa , Q=>Timer_poliv_terrasaQ , ET=>tTimerValue_terrasa_est );
	END_IF
	IF (Modbus.Poliv_terrasa = FALSE ) THEN
		HW_poliv_terrasa	:=	FALSE;
		Timer_poliv_terrasaQ := FALSE;
		Timer_poliv_terrasa(IN:=FALSE , PT:=T#0ms , Q=>Timer_poliv_terrasaQ , ET=>tTimerValue_terrasa_est );
	END_IF
	IF Timer_poliv_terrasa.q THEN
		Modbus.Poliv_terrasa := FALSE;
		HW_poliv_zapad	:=	FALSE;
	END_IF
	
	
	
	IF (Modbus.Poliv_south = TRUE ) THEN
		tTimerValue_south := DINT_TO_TIME(Modbus.Poliv_south_minutes*60*1000);
		HW_poliv_south	:=	TRUE;
		Timer_poliv_south(IN:=NOT Timer_poliv_southQ , PT:=tTimerValue_south , Q=>Timer_poliv_southQ , ET=>tTimerValue_south_est );
	END_IF
	IF (Modbus.Poliv_south = FALSE ) THEN
		HW_poliv_south	:=	FALSE;
		Timer_poliv_southQ := FALSE;
		Timer_poliv_south(IN:=FALSE , PT:=T#0ms , Q=>Timer_poliv_southQ , ET=>tTimerValue_south_est );
	END_IF
	IF Timer_poliv_south.q THEN
		Modbus.Poliv_south := FALSE;
		HW_poliv_south	:=	FALSE;
	END_IF
	
	

	IF (Modbus.Poliv_north = TRUE ) THEN
		tTimerValue_north := DINT_TO_TIME(Modbus.Poliv_north_minutes*60*1000);
		HW_poliv_north	:=	TRUE;
		Timer_poliv_north(IN:=NOT Timer_poliv_northQ , PT:=tTimerValue_north , Q=>Timer_poliv_northQ , ET=>tTimerValue_north_est );
	END_IF
	IF (Modbus.Poliv_north = FALSE ) THEN
		HW_poliv_north	:=	FALSE;
		Timer_poliv_northQ := FALSE;
		Timer_poliv_north(IN:=FALSE , PT:=T#0ms , Q=>Timer_poliv_northQ , ET=>tTimerValue_north_est );
	END_IF
	IF Timer_poliv_north.q THEN
		Modbus.Poliv_north := FALSE;
		HW_poliv_north	:=	FALSE;
	END_IF
	

	IF (Modbus.Poliv_flowers = TRUE ) THEN
		tTimerValue_flowers := DINT_TO_TIME(Modbus.Poliv_flowers_minutes*60*1000);
		HW_poliv_flowers	:=	TRUE;
		Timer_poliv_flowers(IN:=NOT Timer_poliv_flowersQ , PT:=tTimerValue_flowers , Q=>Timer_poliv_flowersQ , ET=>tTimerValue_flowers_est );
	END_IF
	IF (Modbus.Poliv_flowers = FALSE ) THEN
		HW_poliv_flowers	:=	FALSE;
		Timer_poliv_flowersQ := FALSE;
		Timer_poliv_flowers(IN:=FALSE , PT:=T#0ms , Q=>Timer_poliv_flowersQ , ET=>tTimerValue_flowers_est );
	END_IF
	IF Timer_poliv_flowers.q THEN
		Modbus.Poliv_flowers := FALSE;
		HW_poliv_flowers	:=	FALSE;
	END_IF












	



	IF ((HW_poliv_zapad=TRUE OR HW_poliv_terrasa=TRUE 	OR HW_poliv_south =	TRUE OR HW_poliv_north = TRUE) AND (HW_pomp_Garden=FALSE)  )  THEN
		pomp_garden_start			:=TRUE;
	END_IF
	

	TON_pomp_garden(IN := pomp_garden_start, PT:= tTimerValue);
	Modbus.Pomp_garden	 	:= TON_pomp_garden.Q;
	HW_Pomp_garden		:= TON_pomp_garden.Q;
	
	IF (HW_poliv_zapad=FALSE AND HW_poliv_terrasa=FALSE 	AND HW_poliv_south = FALSE  AND HW_poliv_north = FALSE)   THEN
		pomp_garden_start		:= FALSE;
		Modbus.Pomp_garden	 	:= FALSE;
		HW_Pomp_garden		:= FALSE;
	END_IF
ELSE
	HW_poliv_zapad	:=	TRUE;
	HW_poliv_terrasa	:=	TRUE;
	HW_poliv_south 	:=	TRUE;
	HW_poliv_north 	:= 	TRUE;
END_IF
END_PROGRAM

(* POU Power_act, ST *)
PROGRAM Power_act
VAR
	fbCalcSunriseSunset   	: FB_CalcSunriseSunset;
	todSunrise            		: TOD;
   	todSunset          		: TOD;
	dtCurrentDate         		: DT;
	fileTime              		: T_FILETIME;
	fbGetSystemTime       	: GETSYSTEMTIME;
	time_now			: TOD;
	tz					: TIME:=T#5h;
	delta_time			: TIME:=T#2h;

END_VAR
(*
fbGetSystemTime(timeLoDW =>fileTime.dwLowDateTime,
                timeHiDW =>fileTime.dwHighDateTime);
dtCurrentDate:=FILETIME_TO_DT(fileTime);


fbCalcSunriseSunset( fDegreeOfLongitude := 73.26,   (* Longitude of Verl *)
                     fDegreeOfLatitude := 61.15,   (* Latitude of Verl *)
                     fReferenceMeridian := 73.26,  (* Central European Summer Time *)
                     dCurrentDate := DT_TO_DATE(dtCurrentDate),
                     todSunrise => todSunrise,
                     todSunset => todSunset);

time_now	:= DT_TO_TOD(dtCurrentDate)+tz;
*)

IF ((Modbus.Security_status = FALSE  AND Modbus.Sensor_supply = FALSE AND Modbus.Balkon_light_lux < 1000) OR  Modbus.Light_reserv_manual=1 ) THEN
	Modbus.Light_reserv := TRUE;
ELSE
	Modbus.Light_reserv := FALSE;
END_IF

HW_light_rezerv	:=	Modbus.Light_reserv;

(*
IF ( time_now > todSunrise+delta_time  AND  time_now < todSunset-delta_time   ) THEN
		Modbus.Light_reserv := FALSE;
	ELSE
		IF (Modbus.Security_status = FALSE) THEN
			Modbus.Light_reserv := TRUE;
		END_IF
END_IF

IF (Modbus.Security_status = TRUE) THEN
	Modbus.Light_reserv := FALSE;
END_IF



IF (Modbus.Light_reserv=TRUE AND (Modbus.Light_reserv_manual=1 OR Modbus.Light_reserv_manual=2)) THEN
		HW_light_rezerv:=TRUE;
	ELSIF  (Modbus.Light_reserv=TRUE AND  Modbus.Light_reserv_manual=0 ) THEN
		HW_light_rezerv:=FALSE;
	ELSIF (Modbus.Light_reserv=FALSE AND Modbus.Light_reserv_manual=1) THEN
		HW_light_rezerv:=TRUE;
	ELSE
		HW_light_rezerv:=FALSE;
END_IF
*)
END_PROGRAM

(* POU Alarm, ST *)
PROGRAM Alarm
VAR
	alarm						:	 BOOL;
	TRIG_button_alarm			:	R_TRIG;
	TRIG_alarm_smoke_1floor		:	F_TRIG;
	TRIG_alarm_smoke_3floor		:	F_TRIG;
	TRIG_alarm_smoke_drovnik	:	F_TRIG;
	TRIG_alarm_smoke_sklad		:	F_TRIG;
	TRIG_alarm_smoke_stair		:	F_TRIG;

	TRIG_alarm_smoke_sport		:	R_TRIG;
	TRIG_alarm_smoke_2floor		:	R_TRIG;


	TimerValue_alarm				: 	TIME	:=	t#30s;
	Timer_alarm					:	TON;
	Timer_alarm_Q				:	BOOL	:=	FALSE;

	TimerValue_power_smoke		:	 TIME	:=	t#10s;
	Timer_power_smoke			:	TON;
	Timer_power_smoke_Q		:	BOOL	:=	FALSE;

END_VAR
Timer_alarm();
Timer_power_smoke();

IF (SystemTaskInfoArr[1].cycleCount>500)	THEN

	TRIG_alarm_smoke_1floor(CLK :=HW_sensor_smoke_1floor);
	TRIG_alarm_smoke_2floor(CLK :=HW_sensor_smoke_2floor);
	TRIG_alarm_smoke_3floor(CLK :=HW_sensor_smoke_3floor);
	TRIG_alarm_smoke_sport(CLK :=HW_sensor_smoke_sport);
	TRIG_alarm_smoke_sklad(CLK :=HW_sensor_smoke_sklad);
	TRIG_alarm_smoke_drovnik(CLK :=HW_sensor_smoke_drovnik);
	TRIG_alarm_smoke_stair(CLK :=HW_sensor_smoke_stair);



	(*Активируем сирену при сработке датчиков дыма*)
	IF (TRIG_alarm_smoke_1floor.Q OR TRIG_alarm_smoke_2floor.Q OR TRIG_alarm_smoke_3floor.Q OR TRIG_alarm_smoke_sklad.Q OR TRIG_alarm_smoke_stair.Q OR TRIG_alarm_smoke_sport.Q)   THEN
		HW_alarm			:=	1;
		Modbus.Alarm_act	:=	1;
		Timer_alarm(IN:=NOT Timer_alarm_Q , PT:=TimerValue_alarm , Q=>Timer_alarm_Q , ET=> );

		Modbus.Smoke_1floor		:=	TRIG_alarm_smoke_1floor.Q;
		Modbus.Smoke_2floor		:=	TRIG_alarm_smoke_2floor.Q;
		Modbus.Smoke_3floor		:=	TRIG_alarm_smoke_3floor.Q;
		Modbus.Smoke_sklad		:=	TRIG_alarm_smoke_sklad.Q;
		Modbus.Smoke_drovnik	:=	TRIG_alarm_smoke_drovnik.Q;
		Modbus.Smoke_stair		:=	TRIG_alarm_smoke_stair.Q;


	END_IF

	TRIG_button_alarm(CLK :=HW_button_alarm);


	(*Обработка нажатия кнопки Сирена *)
	IF (TRIG_button_alarm.Q) THEN
		(*Если отключаем  сирену *)
		IF (Modbus.Alarm_act = 1)	THEN
			Modbus.Alarm_act	:=	0;
			HW_alarm			:=	0;
			HW_power_smoke_sen:=1;  (*отключаем питание датчиков на 3 секунды для сброса сигнала тревоги*)
			Timer_power_smoke(IN:=NOT Timer_power_smoke_Q , PT:=TimerValue_power_smoke , Q=>Timer_power_smoke_Q , ET=> );
			(*Иначе - включаем, независимо от показаний датчиков *)
		ELSE
			Modbus.Alarm_act	:=	1;
			HW_alarm			:=	1;
			Timer_alarm(IN:=NOT Timer_alarm_Q , PT:=TimerValue_alarm , Q=>Timer_alarm_Q , ET=> );
		END_IF
	END_IF (*Конец обработки нажатия кнопки *)

	(*Время активности сирены и действия по окончании таймера сирены*)
	IF Timer_alarm.Q THEN

		Modbus.Smoke_1floor		:=	FALSE;
		Modbus.Smoke_2floor		:=	FALSE;
		Modbus.Smoke_3floor		:=	FALSE;
		Modbus.Smoke_sklad		:=	FALSE;
		Modbus.Smoke_drovnik	:=	FALSE;
		Modbus.Smoke_stair		:=	FALSE;


		Modbus.Alarm_act		:=	0;
		HW_alarm				:=	0;
		HW_power_smoke_sen	:=	1;
		Timer_alarm_Q := FALSE;
		Timer_alarm(IN:=FALSE , PT:=T#0ms , Q=>Timer_alarm_Q , ET=> );
		Timer_power_smoke(IN:=NOT Timer_power_smoke_Q , PT:=TimerValue_power_smoke , Q=>Timer_power_smoke_Q , ET=> );
	END_IF

	(*Включение питаня датчиков *)
	IF Timer_power_smoke.Q THEN
		HW_power_smoke_sen := 0;
		Timer_power_smoke_Q := FALSE;
		Timer_power_smoke(IN:=FALSE , PT:=T#0ms , Q=>Timer_power_smoke_Q , ET=> );
	END_IF

END_IF
END_PROGRAM

(* POU Buttons, ST *)
PROGRAM Buttons
VAR
(*	TRIG_BUT_light1			:	R_TRIG;
	TRIG_BUT_light_kitchen	:	R_TRIG;
	TRIG_BUT_light_terrasa	:	R_TRIG;
*)
	SW_LIGHT_GARDEN			: SM_BUTT;		(* вкл/откл прожектор *)
	SW_VOROTA				: FB_ShortLongClick;
	TRIG_vorota_open			: R_TRIG;
	TRIG_vorota_modbus			: R_TRIG;
	TRIG_vorota_open_modbus	: R_TRIG;
(*	SW_VOROTA				: SM_BUTT; *)

(*	Vorota_switch					: BOOL:=FALSE; *)
	Vorota_open					: BOOL:=FALSE;

	Pulse						: TP;
	PT_length					: TIME:= T#500ms;


	Timer_vo					: TON;
	Timer_voQ					: BOOL;
	tTimerValue_vo				: TIME:= T#23500ms;





END_VAR
	SW_LIGHT_GARDEN		(IN:=HW_button_light_garden, IN1:=Modbus.Light_garden, 	Q=>Modbus.Light_garden);		(* Конпка *)
	SW_VOROTA			(bSwitch :=HW_button_vorota, tSwitchTime   := t#2000ms);

	iobroker.Vorota_active:=FALSE;
	Timer_vo();

	TRIG_vorota_modbus(CLK :=Modbus.Vorota);
	TRIG_vorota_open_modbus(CLK :=Modbus.Vorota_open);

	IF TRIG_vorota_modbus.Q		THEN
		Pulse (IN:=TRUE, PT:=PT_length, Q=>HW_vorota , ET=> );
	END_IF

	Pulse (IN:=SW_VOROTA.bShortClick, PT:=PT_length, Q=>HW_vorota , ET=> );

(*	HW_vorota					:=	Modbus.Vorota; *)

	IF (SW_VOROTA.bShortClick) THEN
		iobroker.Vorota_active:=TRUE;
	END_IF




	IF (SW_VOROTA.bLongClick OR TRIG_vorota_open_modbus.Q) THEN
		Vorota_open				:= TRUE;
		iobroker.Vorota_open_active:=TRUE;
	END_IF

	Pulse (IN:=SW_VOROTA.bLongClick, PT:=PT_length, Q=>HW_vorota , ET=> );
	Pulse (IN:=TRIG_vorota_open_modbus.Q, PT:=PT_length, Q=>HW_vorota , ET=> );

	IF 	Vorota_open		THEN
		Timer_vo(IN:=NOT Timer_voQ , PT:=tTimerValue_vo , Q=>Timer_voQ , ET=> );
	END_IF

	TRIG_vorota_open(CLK :=Timer_voQ);

	IF TRIG_vorota_open.Q		THEN
		Pulse (IN:=TRUE, PT:=PT_length, Q=>HW_vorota , ET=> );
		Vorota_open				:= FALSE;
		iobroker.Vorota_open_active:=FALSE;
	END_IF
END_PROGRAM

(* POU SM_BUTT, ST *)
FUNCTION_BLOCK SM_BUTT            (* ФУНКЦИОНАЛЬНЫЙ БЛОК ДЛЯ ПРОСТОЙ КНОПКИ *)
    VAR_INPUT
       	IN: BOOL;          	(*ВХОД ЗА КОТОРЫМ МЫ СЛЕДИМ *)
	IN1:BOOL;				(*ВЫХОД ЗА КОТОРЫМ ТОЖЕ СЛЕДИМ*)
    END_VAR

    VAR_OUTPUT
	Q : BOOL;        			(*СОСТОЯНИЕ ВЫХОДА*)
    END_VAR
    VAR
  MEM : BOOL;    			(* ВНУТРЕННЯЯ ПЕРЕМЕННАЯ ДЛЯ ХРАНЕНИЯ СОСТОЯНИЯ КНОПКИ *)
    END_VAR
Q:=IN1;

IF IN AND NOT MEM THEN 	(* ПОЙМАЛИ ПЕРЕДНИЙ ФРОНТ - НАЖАЛИ НА КНОПКУ *)
	Q := NOT IN1;    			(* МЕНЯЕМ СОСТОЯНИЕ ВЫХОДА НА ПРОТИВОПОЛОЖНОЕ *)
END_IF

MEM := IN;                       		(* ЗАПОМИНАЕМ ТЕКУЩЕЕ ЗНАЧЕНИЕ КНОПКИ *)
END_FUNCTION_BLOCK

(* POU ParnikWindowCtrl, ST *)
PROGRAM ParnikWindowCtrl
VAR
    (* Modbus I/O (использовать точно как заданы) *)
    (* Modbus.Street_temp : REAL *)
    (* Modbus.Parnik_set_temp_street_min : REAL *)
    (* Modbus.Parnik_air_temp : REAL *)
    (* Modbus.Parnik_set_auto_window : BOOL *)
    (* Modbus.Parnik_current_level_window : UINT *) (* 0=closed,1=30%,2=60%,3=100% *)
    (* Modbus.Parnik_manual_level_window : UINT *)
    (* Modbus.Parnik_temp_step1_window : UINT *) (* threshold for 30% *)
    (* Modbus.Parnik_temp_step2_window : UINT *) (* threshold for 60% *)

    (* HW outputs *)
    (* HW_power_supply_parnik : BOOL *)
    (* HW_power_polarity_parnik : BOOL *)

    (* Internal *)
    closeTON : TON;                 (* PT = 60s *)
    openTON  : TON;                 (* PT = variable *)
    state : UINT := 0;              (* 0=idle,1=closing,2=opening *)
    targetLevel : UINT := 0;        (* desired final level 0..3 *)
    openTime : TIME := T#0s;
    hysteresis : REAL := 3.0;
    prevManualLevel : UINT := 255;
    manualReq : BOOL := FALSE;
    startClose : BOOL := FALSE;
    startOpen  : BOOL := FALSE;
    firstScan : BOOL := TRUE;
    trigLevel1,trigLevel2,trigLevel3 : BOOL;

END_VAR
hysteresis		:=	3.0;

IF firstScan THEN
    Modbus.Parnik_current_level_window := 0; (* default closed *)
    
    (* Исправлено: Защита старта теперь сразу взводит триггеры *)
    IF Modbus.Parnik_air_temp > (INT_TO_REAL(Modbus.Parnik_temp_step1_window) - hysteresis)
       AND Modbus.Parnik_air_temp < (INT_TO_REAL(Modbus.Parnik_temp_step1_window) + hysteresis) THEN
        targetLevel := 1;
        trigLevel1 := TRUE;
        trigLevel2 := FALSE;
    ELSE
        targetLevel := 0;
        trigLevel1 := FALSE;
        trigLevel2 := FALSE;
    END_IF;

    HW_power_supply_parnik := FALSE;
    HW_power_polarity_parnik := FALSE;
    closeTON(IN := FALSE, PT := T#60s);
    openTON(IN := FALSE, PT := T#60s);
    prevManualLevel := Modbus.Parnik_manual_level_window;
    firstScan := FALSE;
END_IF;

(* Определение ручного запроса *)
manualReq := FALSE;
IF NOT Modbus.Parnik_set_auto_window THEN
    IF Modbus.Parnik_manual_level_window <> prevManualLevel THEN
        manualReq := TRUE;
    END_IF;
END_IF;
prevManualLevel := Modbus.Parnik_manual_level_window;

(* Determine targetLevel according to requested logic *)
IF Modbus.Parnik_set_auto_window THEN
    (* AUTO - Чистая логика RS-триггеров *)
    
    (* УЛИЦА: Если на улице слишком холодно, принудительно закрываем всё *)
    IF Modbus.Street_temp < Modbus.Parnik_set_temp_street_min THEN
        targetLevel := 0;
        
    ELSE
        (* РАБОТА ПО ТЕМПЕРАТУРЕ ВНУТРИ *)
        
        (* Триггер Уровня 2 *)
        IF Modbus.Parnik_air_temp > (INT_TO_REAL(Modbus.Parnik_temp_step2_window) + hysteresis) THEN
            trigLevel2 := TRUE;
        ELSIF Modbus.Parnik_air_temp < (INT_TO_REAL(Modbus.Parnik_temp_step2_window) - hysteresis) THEN
            trigLevel2 := FALSE;
        END_IF;

        (* Триггер Уровня 1 *)
        IF Modbus.Parnik_air_temp > (INT_TO_REAL(Modbus.Parnik_temp_step1_window) + hysteresis) THEN
            trigLevel1 := TRUE;
        ELSIF Modbus.Parnik_air_temp < (INT_TO_REAL(Modbus.Parnik_temp_step1_window) - hysteresis) THEN
            trigLevel1 := FALSE;
        END_IF;

        (* Расстановка приоритетов уровней *)
        IF trigLevel2 THEN
            targetLevel := 2;
        ELSIF trigLevel1 THEN
            targetLevel := 1;
        ELSE
            targetLevel := 0;
        END_IF;

    END_IF;

ELSE
    (* MANUAL - независимый от температуры режим *)
    CASE Modbus.Parnik_manual_level_window OF
        0: targetLevel := 0;
        1: targetLevel := 1;
        2: targetLevel := 2;
        3: targetLevel := 3;
        ELSE targetLevel := Modbus.Parnik_current_level_window;
    END_CASE;
END_IF;

(* Force sequence restart if manual request detected while in idle *)
IF manualReq AND (state = 0) THEN
    Modbus.Parnik_current_level_window := 99; 
END_IF;

(* State Machine Trigger (when Idle) *)
IF state = 0 THEN
    startClose := FALSE;
    startOpen := FALSE;
    
    IF Modbus.Parnik_current_level_window <> targetLevel THEN
        
        IF targetLevel = 0 THEN
            (* Полное закрытие *)
            startClose := TRUE;
            state := 1;
        ELSIF Modbus.Parnik_current_level_window = 99 THEN
            (* Сброс по ручной команде -> сначала закрываем до упора *)
            startClose := TRUE;
            state := 1;
        ELSE
            (* Движение к уровню > 0 *)
            IF targetLevel > Modbus.Parnik_current_level_window AND Modbus.Parnik_current_level_window <> 0 THEN
                (* ДВИЖЕНИЕ ВВЕРХ БЕЗ ЗАКРЫТИЯ (Рассчитываем дельту) *)
                IF Modbus.Parnik_current_level_window = 1 AND targetLevel = 2 THEN openTime := T#25s;
                ELSIF Modbus.Parnik_current_level_window = 1 AND targetLevel = 3 THEN openTime := T#55s;
                ELSIF Modbus.Parnik_current_level_window = 2 AND targetLevel = 3 THEN openTime := T#30s;
                ELSE openTime := T#0s;
                END_IF;

                IF openTime > T#0s THEN
                    startOpen := TRUE;
                    state := 2;
                ELSE
                    Modbus.Parnik_current_level_window := targetLevel;
                END_IF;
            ELSE
                (* ДВИЖЕНИЕ ВНИЗ ИЛИ СТАРТ ИЗ НУЛЯ -> сначала полное закрытие для точности *)
                startClose := TRUE;
                state := 1;
            END_IF;
        END_IF;
    END_IF;
END_IF;

(* State machine *)
CASE state OF
    0: (* Idle *)
        HW_power_supply_parnik := FALSE;
        HW_power_polarity_parnik := FALSE;
        
    1: (* Closing (60s) *)
        closeTON(IN := startClose, PT := T#60s);
        HW_power_polarity_parnik := FALSE; (* False = закрытие *)
        HW_power_supply_parnik := startClose;

        IF closeTON.Q THEN
            closeTON(IN := FALSE, PT := T#60s);
            startClose := FALSE;
            HW_power_supply_parnik := FALSE;
            Modbus.Parnik_current_level_window := 0; (* Окно гарантированно в нулю *)
            
            IF targetLevel > 0 THEN
                (* Расчет чистого времени открытия ИЗ НУЛЯ *)
                CASE targetLevel OF
                    1: openTime := T#5s;
                    2: openTime := T#30s;
                    3: openTime := T#60s;
                    ELSE openTime := T#0s;
                END_CASE;

                IF openTime > T#0s THEN
                    startOpen := TRUE;
                    state := 2;
                ELSE
                    Modbus.Parnik_current_level_window := targetLevel;
                    state := 0;
                END_IF;
            ELSE
                state := 0;
            END_IF;
        END_IF;

    2: (* Opening *)
        openTON(IN := startOpen, PT := openTime);
        HW_power_polarity_parnik := TRUE; (* True = открытие *)
        HW_power_supply_parnik := startOpen;

        IF openTON.Q THEN
            openTON(IN := FALSE, PT := openTime);
            startOpen := FALSE;
            HW_power_supply_parnik := FALSE;
            Modbus.Parnik_current_level_window := targetLevel; (* Установка финального статуса *)
            state := 0;
        END_IF;

ELSE
    HW_power_supply_parnik := FALSE;
    startClose := FALSE;
    startOpen := FALSE;
    closeTON(IN := FALSE, PT := T#60s);
    openTON(IN := FALSE, PT := T#60s);
    state := 0;
END_CASE;
END_PROGRAM

(* POU Parnik_heat, ST *)
PROGRAM Parnik_heat
VAR
	(* Настройки логики *)
	rAirStartOutside : REAL; (* Порог включения по улице вечером *)
	rWaterMaxLimit   : REAL := 35.0; (* Верхний лимит воды в трубе *)
	rWaterMinLimit   : REAL := 30.0; (* Нижний лимит воды в трубе ночью *)
	
	(* Внутренние флаги *)
	bNightModeActive : BOOL; (* Разрешение на работу ночного подогрева *)

	dtCurrentDate         		: DT;
	fileTime              		: T_FILETIME;
	fbGetSystemTime       	: GETSYSTEMTIME;
	time_now			: TOD;
	tz					: TIME:=T#5h;
	test1, test2, test3 ,hours,minutes		: INT;
	hm				:ExtractTime;

END_VAR
rAirStartOutside	:= Modbus.Parnik_temp_step1_window-1;

fbGetSystemTime(timeLoDW =>fileTime.dwLowDateTime,
                timeHiDW =>fileTime.dwHighDateTime);
dtCurrentDate:=FILETIME_TO_DT(fileTime);
time_now	:= DT_TO_TOD(dtCurrentDate)+tz;

hm(tm:=time_now, h=>hours, m=>minutes);


(* АКТИВАЦИЯ НОЧНОГО РЕЖИМА ОПЕРЕЖЕНИЕ И ЧАСЫ *)
(* Включение: на улице холоднее +10 и время между 12:00 дня и 06:00 утра *)
IF (Modbus.Parnik_air_temp <= rAirStartOutside) AND (hours >= 12 OR hours < 6) THEN
	bNightModeActive := TRUE;
END_IF;

(* Гарантированное выключение: наступило 06:00 утра ИЛИ на улице потеплело выше +12 *)
IF (hours >= 6 AND hours < 12) OR (Modbus.Parnik_air_temp > (rAirStartOutside + 2.0)) THEN
	bNightModeActive := FALSE;
END_IF;


(* УПРАВЛЕНИЕ ГРЕЮЩИМ КАБЕЛЕМ ПО ТЕМПЕРАТУРЕ ВОДЫ *)
IF bNightModeActive THEN
	
	(* Двухпозиционное регулирование с гистерезисом по воде в трубе *)
	IF Modbus.Parnik_pipe_temp >= rWaterMaxLimit THEN
		HW_parnik_heat := FALSE; (* Выключаем подогрев при +35 *)
	ELSIF Modbus.Parnik_pipe_temp <= rWaterMinLimit THEN
		HW_parnik_heat := TRUE;  (* Включаем подогрев при +30 *)
	END_IF;
	
ELSE
	
	(* Днем или после 6 утра принудительно отключаем нагрев *)
	HW_parnik_heat := FALSE;

END_IF;

Modbus.Teplica_DO8	:=	HW_parnik_heat;
END_PROGRAM

(* POU Light_balkon_rassada, ST *)
PROGRAM Light_balkon_rassada
VAR

	gisterezis		: REAL:=1000; (*Гистерезис включения подсветки *)

END_VAR
(*LIGHT BALKON RASSADA *)
IF (HW_light_rassada = FALSE) THEN

	IF (Modbus.Balkon_light_rassada_allow=FALSE OR Modbus.Balkon_light_lux> Modbus.Teplica_light_set_low+gisterezis ) THEN
		HW_light_rassada:=FALSE;
	END_IF

	IF (Modbus.Balkon_light_rassada_allow= TRUE AND (Modbus.Balkon_light_lux <  Modbus.Teplica_light_set_low-gisterezis ) ) THEN
		HW_light_rassada:=TRUE;
	END_IF
END_IF


IF (HW_light_rassada = TRUE) THEN

	IF (Modbus.Balkon_light_rassada_allow=FALSE OR Modbus.Balkon_light_lux-Modbus.Balkon_power_light_lux> Modbus.Teplica_light_set_low+gisterezis ) THEN
		HW_light_rassada:=FALSE;
	END_IF

	IF (Modbus.Balkon_light_rassada_allow= TRUE AND (Modbus.Balkon_light_lux-Modbus.Balkon_power_light_lux <  Modbus.Teplica_light_set_low-gisterezis ) ) THEN
		HW_light_rassada:=TRUE;
	END_IF
END_IF
END_PROGRAM

(* POU Mqtt, ST *)
PROGRAM Mqtt
VAR
	FB_Mqtt_Controller 		: FB_Mqtt_Controller_V10;
	stMqttSettings				: ST_MqttSettings;
	bMqttControllerBusy		: BOOL;

	FB_Mqtt_Publish1 			: FB_Mqtt_Publish_V10;
	FB_Mqtt_Publish2			: FB_Mqtt_Publish_V10;
	FB_Mqtt_Publish3			: FB_Mqtt_Publish_V10;
	FB_Mqtt_Publish4			: FB_Mqtt_Publish_V10;
	FB_Mqtt_Publish5			: FB_Mqtt_Publish_V10;
	FB_Mqtt_Publish6			: FB_Mqtt_Publish_V10;
	FB_Mqtt_Publish7			: FB_Mqtt_Publish_V10;
	FB_Mqtt_Publish8			: FB_Mqtt_Publish_V10;
	FB_Mqtt_Publish9			: FB_Mqtt_Publish_V10;
	FB_Mqtt_Publish10		: FB_Mqtt_Publish_V10;
	FB_Mqtt_Publish11		: FB_Mqtt_Publish_V10;
	FB_Mqtt_Publish12		: FB_Mqtt_Publish_V10;
	FB_Mqtt_Publish13 		: FB_Mqtt_Publish_V10;
	FB_Mqtt_Publish14		: FB_Mqtt_Publish_V10;
	FB_Mqtt_Publish15		: FB_Mqtt_Publish_V10;
	FB_Mqtt_Publish16		: FB_Mqtt_Publish_V10;
	FB_Mqtt_Publish17		: FB_Mqtt_Publish_V10;
	FB_Mqtt_Publish18		: FB_Mqtt_Publish_V10;
	FB_Mqtt_Publish19		: FB_Mqtt_Publish_V10;
	FB_Mqtt_Publish20		: FB_Mqtt_Publish_V10;
	FB_Mqtt_Publish21		: FB_Mqtt_Publish_V10;
	FB_Mqtt_Publish22		: FB_Mqtt_Publish_V10;
	FB_Mqtt_Publish23		: FB_Mqtt_Publish_V10;
	FB_Mqtt_Publish24		: FB_Mqtt_Publish_V10;
	FB_Mqtt_Publish25		: FB_Mqtt_Publish_V10;
	FB_Mqtt_Publish26		: FB_Mqtt_Publish_V10;
	FB_Mqtt_Publish27		: FB_Mqtt_Publish_V10;
	FB_Mqtt_Publish28		: FB_Mqtt_Publish_V10;

	bPublishBusy1			: BOOL;
	bPublishBusy2			: BOOL;
	bPublishBusy3			: BOOL;
	bPublishBusy4			: BOOL;
	bPublishBusy5			: BOOL;
	bPublishBusy6			: BOOL;
	bPublishBusy7			: BOOL;
	bPublishBusy8			: BOOL;
	bPublishBusy9			: BOOL;
	bPublishBusy10			: BOOL;
	bPublishBusy11			: BOOL;
	bPublishBusy12			: BOOL;
	bPublishBusy13			: BOOL;
	bPublishBusy14			: BOOL;
	bPublishBusy15			: BOOL;
	bPublishBusy16			: BOOL;
	bPublishBusy17			: BOOL;
	bPublishBusy18			: BOOL;
	bPublishBusy19			: BOOL;
	bPublishBusy20			: BOOL;
	bPublishBusy21			: BOOL;
	bPublishBusy22			: BOOL;
	bPublishBusy23			: BOOL;
	bPublishBusy24			: BOOL;
	bPublishBusy25			: BOOL;
	bPublishBusy26			: BOOL;
	bPublishBusy27			: BOOL;
	bPublishBusy28			: BOOL;

	START: BOOL;
END_VAR
FB_Mqtt_Controller (
		bActive			:= TRUE,
		sMqttClientId		:= 'plc',
		sMqttUserId		:= 'mqtt',
		sMqttPassword	:= 'mqtt',
		sMqttBrokerIp		:= '192.168.2.200',
		nMqttBrokerPort	:= 1883,
		stMqttSettings		:= stMqttSettings,
		bBusy			=> bMqttControllerBusy
	);

IF NOT bMqttControllerBusy THEN

	FB_Mqtt_Publish1(sTopic:='BECKHOFF_CX9000/Mercury/M1T1',sValue:=REAL_TO_STRING(Mercury.M1T1),bRetain:=FALSE, stMqttSettings:=stMqttSettings,bBusy => bPublishBusy1 );
	FB_Mqtt_Publish2(sTopic:='BECKHOFF_CX9000/Mercury/M1T2',sValue:=REAL_TO_STRING(Mercury.M1T2),bRetain:=FALSE, stMqttSettings:=stMqttSettings,bBusy => bPublishBusy2 );
	FB_Mqtt_Publish3(sTopic:='BECKHOFF_CX9000/Mercury/M2T1',sValue:=REAL_TO_STRING(Mercury.M2T1),bRetain:=FALSE, stMqttSettings:=stMqttSettings,bBusy => bPublishBusy3 );
	FB_Mqtt_Publish4(sTopic:='BECKHOFF_CX9000/Mercury/M2T2',sValue:=REAL_TO_STRING(Mercury.M2T2),bRetain:=FALSE, stMqttSettings:=stMqttSettings,bBusy => bPublishBusy4 );
	FB_Mqtt_Publish5(sTopic:='BECKHOFF_CX9000/Mercury/M3T1',sValue:=REAL_TO_STRING(Mercury.M3T1),bRetain:=FALSE, stMqttSettings:=stMqttSettings,bBusy => bPublishBusy5 );
	FB_Mqtt_Publish6(sTopic:='BECKHOFF_CX9000/Mercury/M3T2',sValue:=REAL_TO_STRING(Mercury.M3T2),bRetain:=FALSE, stMqttSettings:=stMqttSettings,bBusy => bPublishBusy6 );
	FB_Mqtt_Publish7(sTopic:='BECKHOFF_CX9000/Mercury/M4T1',sValue:=REAL_TO_STRING(Mercury.M4T1),bRetain:=FALSE, stMqttSettings:=stMqttSettings,bBusy => bPublishBusy7 );
	FB_Mqtt_Publish8(sTopic:='BECKHOFF_CX9000/Mercury/M4T2',sValue:=REAL_TO_STRING(Mercury.M4T2),bRetain:=FALSE, stMqttSettings:=stMqttSettings,bBusy => bPublishBusy8 );
	FB_Mqtt_Publish9(sTopic:='BECKHOFF_CX9000/Mercury/M5T1',sValue:=REAL_TO_STRING(Mercury.M5T1),bRetain:=FALSE, stMqttSettings:=stMqttSettings,bBusy => bPublishBusy9 );
	FB_Mqtt_Publish10(sTopic:='BECKHOFF_CX9000/Mercury/M5T2',sValue:=REAL_TO_STRING(Mercury.M5T2),bRetain:=FALSE, stMqttSettings:=stMqttSettings,bBusy => bPublishBusy10 );
	FB_Mqtt_Publish11(sTopic:='BECKHOFF_CX9000/Mercury/M6T1',sValue:=REAL_TO_STRING(Mercury.M6T1),bRetain:=FALSE, stMqttSettings:=stMqttSettings,bBusy => bPublishBusy11 );
	FB_Mqtt_Publish12(sTopic:='BECKHOFF_CX9000/Mercury/M6T2',sValue:=REAL_TO_STRING(Mercury.M6T2),bRetain:=FALSE, stMqttSettings:=stMqttSettings,bBusy => bPublishBusy12 );
	FB_Mqtt_Publish13(sTopic:='BECKHOFF_CX9000/Mercury/M7T1',sValue:=REAL_TO_STRING(Mercury.M7T1),bRetain:=FALSE, stMqttSettings:=stMqttSettings,bBusy => bPublishBusy13 );
	FB_Mqtt_Publish14(sTopic:='BECKHOFF_CX9000/Mercury/M7T2',sValue:=REAL_TO_STRING(Mercury.M7T2),bRetain:=FALSE, stMqttSettings:=stMqttSettings,bBusy => bPublishBusy14);
	FB_Mqtt_Publish15(sTopic:='BECKHOFF_CX9000/Mercury/M8T1',sValue:=REAL_TO_STRING(Mercury.M8T1),bRetain:=FALSE, stMqttSettings:=stMqttSettings,bBusy => bPublishBusy15 );
	FB_Mqtt_Publish16(sTopic:='BECKHOFF_CX9000/Mercury/M8T2',sValue:=REAL_TO_STRING(Mercury.M8T2),bRetain:=FALSE, stMqttSettings:=stMqttSettings,bBusy => bPublishBusy16 );
	FB_Mqtt_Publish17(sTopic:='BECKHOFF_CX9000/Mercury/M9T1',sValue:=REAL_TO_STRING(Mercury.M9T1),bRetain:=FALSE, stMqttSettings:=stMqttSettings,bBusy => bPublishBusy17 );
	FB_Mqtt_Publish18(sTopic:='BECKHOFF_CX9000/Mercury/M9T2',sValue:=REAL_TO_STRING(Mercury.M9T2),bRetain:=FALSE, stMqttSettings:=stMqttSettings,bBusy => bPublishBusy18 );
	FB_Mqtt_Publish19(sTopic:='BECKHOFF_CX9000/Mercury/M10T1',sValue:=REAL_TO_STRING(Mercury.M10T1),bRetain:=FALSE, stMqttSettings:=stMqttSettings,bBusy => bPublishBusy19 );
	FB_Mqtt_Publish20(sTopic:='BECKHOFF_CX9000/Mercury/M10T2',sValue:=REAL_TO_STRING(Mercury.M10T2),bRetain:=FALSE, stMqttSettings:=stMqttSettings,bBusy => bPublishBusy20 );
	FB_Mqtt_Publish21(sTopic:='BECKHOFF_CX9000/Mercury/M11T1',sValue:=REAL_TO_STRING(Mercury.M11T1),bRetain:=FALSE, stMqttSettings:=stMqttSettings,bBusy => bPublishBusy21 );
	FB_Mqtt_Publish22(sTopic:='BECKHOFF_CX9000/Mercury/M11T2',sValue:=REAL_TO_STRING(Mercury.M11T2),bRetain:=FALSE, stMqttSettings:=stMqttSettings,bBusy => bPublishBusy22 );
	FB_Mqtt_Publish23(sTopic:='BECKHOFF_CX9000/Mercury/M12T1',sValue:=REAL_TO_STRING(Mercury.M12T1),bRetain:=FALSE, stMqttSettings:=stMqttSettings,bBusy => bPublishBusy23 );
	FB_Mqtt_Publish24(sTopic:='BECKHOFF_CX9000/Mercury/M12T2',sValue:=REAL_TO_STRING(Mercury.M12T2),bRetain:=FALSE, stMqttSettings:=stMqttSettings,bBusy => bPublishBusy24 );
	FB_Mqtt_Publish25(sTopic:='BECKHOFF_CX9000/Sensors/Control_hum',sValue:=REAL_TO_STRING(iob_mqtt.Control_hum),bRetain:=FALSE, stMqttSettings:=stMqttSettings,bBusy => bPublishBusy25 );
	FB_Mqtt_Publish26(sTopic:='BECKHOFF_CX9000/Sensors/Control_temp',sValue:=REAL_TO_STRING(iob_mqtt.Control_temp),bRetain:=FALSE, stMqttSettings:=stMqttSettings,bBusy => bPublishBusy26 );
	FB_Mqtt_Publish27(sTopic:='BECKHOFF_CX9000/Sensors/Control_hum2',sValue:=REAL_TO_STRING(iob_mqtt.Control_hum2),bRetain:=FALSE, stMqttSettings:=stMqttSettings,bBusy => bPublishBusy27 );
	FB_Mqtt_Publish28(sTopic:='BECKHOFF_CX9000/Sensors/Control_temp2',sValue:=REAL_TO_STRING(iob_mqtt.Control_temp2),bRetain:=FALSE, stMqttSettings:=stMqttSettings,bBusy => bPublishBusy28 );

END_IF
(*    END    SEND DATA VIA MQTT  *)
END_PROGRAM

(* POU FB_Mqtt_Controller_V10, ST *)
(* @NESTEDCOMMENTS := 'Yes' *)
(* @PATH := '\/_Generic\/Mqtt' *)
(* @OBJECTFLAGS := '0, 8' *)
(* @SYMFILEFLAGS := '2048' *)
FUNCTION_BLOCK FB_Mqtt_Controller_V10
VAR_INPUT
(*	bActive			: BOOL := FALSE;
	sMqttClientId	: STRING[23]:='plc';
	sMqttUserId	: STRING[25] := 'mqtt';
	sMqttPassword	: STRING[25] := 'mqtt';
	sMqttBrokerIP	: STRING[15]:='192.168.3.200';
	nMqttBrokerPort	: UDINT := 1883;
*)
	bActive			: BOOL := FALSE;
	sMqttClientId	: STRING[23];
	sMqttUserId	: STRING[25] := '';
	sMqttPassword	: STRING[25] := '';
	sMqttBrokerIP	: STRING[15];
	nMqttBrokerPort	: UDINT := 1883;
END_VAR
VAR_OUTPUT
	bBusy	: BOOL := FALSE;
END_VAR
VAR_IN_OUT
	stMqttSettings	: ST_MqttSettings;
END_VAR
VAR
	iState			: INT := 0;
	fbSocketConnect	: FB_SocketConnect;
	fbSocketClose	: FB_SocketClose;

	fbMqttTelegramConnect	: FB_MqttTelegram_Connect_V10;
	fbMqttTelegramPingReq	: FB_MqttTelegram_PingReq_V10;
	fbMqttSend				: FB_Mqtt_Send_V10;
	fbMqttReceive			: FB_Mqtt_Receive_V10;
END_VAR
VAR CONSTANT
	C_STARTUP					: INT := 0;
	C_CONNECT					: INT := 100;
	C_CONNECT_WAIT				: INT := 110;
	C_CLOSE						: INT := 200;
	C_CLOSE_WAIT				: INT := 210;
	C_IDLE						: INT := 500;
END_VAR
(* @END_DECLARATION := '0' *)
(*
 * Connects to mqtt broker
 * Sends connect message
 * Sends ping(back)
 * Sends disconnect
 *)
CASE iState OF
	C_STARTUP:
		stMqttSettings.bConnected			:= FALSE;
		stMqttSettings.bConnectPackageSent	:= FALSE;
		stMqttSettings.bDisconnect			:= FALSE;
		stMqttSettings.bSocketConnection	:= FALSE;
		stMqttSettings.bError				:= FALSE;
		stMqttSettings.bValidConnection		:= FALSE;
		stMqttSettings.wPackageIdentifier	:= 1;
		stMqttSettings.bActive				:= bActive;
		stMqttSettings.hSocket				:= fbSocketConnect.hSocket;
		stMqttSettings.nMqttBrokerPort		:= nMqttBrokerPort;
		stMqttSettings.sMqttBrokerIP		:= sMqttBrokerIP;
		stMqttSettings.sMqttClientId		:= sMqttClientId;
		stMqttSettings.sMqttUserId		:= sMqttUserId;
		stMqttSettings.sMqttPassword		:= sMqttPassword;

		stMqttSettings.stMqttReceivedTelegram.nDataLength := 0;

		bBusy := FALSE;

		CallMqttBlocks();

		IF bActive THEN
			iState := C_CONNECT;
		END_IF;

	(* Start connection *)
	C_CONNECT:
		bBusy := TRUE;

		fbSocketConnect(
			bExecute	:= FALSE
		);

		fbSocketConnect(
			sSrvNetId	:= '',
			sRemoteHost	:= sMqttBrokerIP,
			nRemotePort	:= nMqttBrokerPort,
			bExecute	:= TRUE,
			tTimeout	:= USINT_TO_TIME(stMqttSettings.usKeepAliveTime) + t#10s
		);

		iState := C_CONNECT_WAIT;

	(* Wait till connected *)
	C_CONNECT_WAIT:
		fbSocketConnect(
			bExecute := FALSE
		);

		IF
			NOT fbSocketConnect.bBusy
			AND NOT fbSocketConnect.bError
		THEN
			iState 								:= C_IDLE;
			stMqttSettings.hSocket				:= fbSocketConnect.hSocket;
			stMqttSettings.bSocketConnection	:= TRUE;
		END_IF;

		IF fbSocketConnect.bError THEN
			iState := C_STARTUP;
		END_IF;

		IF NOT stMqttSettings.bActive THEN
			iState := C_STARTUP;
		END_IF;

	(* Close connection *)
	C_CLOSE:
		bBusy := TRUE;

		fbSocketClose(
			bExecute	:= TRUE,
			hSocket		:= stMqttSettings.hSocket
		);

		iState := C_CLOSE_WAIT;

	(* Wait close connection *)
	C_CLOSE_WAIT:
		fbSocketClose(
			bExecute := FALSE
		);

		IF
			NOT fbSocketClose.bBusy
			AND NOT fbSocketClose.bError
		THEN
			iState := C_STARTUP;
		END_IF;

		IF fbSocketClose.bError THEN
			iState := C_STARTUP;
		END_IF;

		IF NOT stMqttSettings.bActive THEN
			iState := C_STARTUP;
		END_IF;

	(* Idle *)
	C_IDLE:
		bBusy 					:= FALSE;
		stMqttSettings.bActive	:= bActive;

		stMqttSettings.bValidConnection :=
			NOT stMqttSettings.bError
			AND NOT stMqttSettings.bDisconnect
			AND stMqttSettings.bConnected
			AND stMqttSettings.bSocketConnection
			AND stMqttSettings.bActive;

		CallMqttBlocks();

		IF
			stMqttSettings.bDisconnect
			OR stMqttSettings.bError
			OR NOT stMqttSettings.bActive
		THEN
			IF
				stMqttSettings.bConnected
				OR stMqttSettings.bSocketConnection
			THEN
				(* TODO : send disconnect *)
				iState := C_CLOSE;
			ELSE
				iState := C_CLOSE;
			END_IF;
		END_IF;

	ELSE
		iState := C_STARTUP;
END_CASE;
(*	END_FUNCTION_BLOCK	*)
END_FUNCTION_BLOCK
ACTION CallMqttBlocks:
(*ACTION	CallMqttBlocks: *)
fbMqttReceive(
	stMqttSettings := stMqttSettings
);

fbMqttTelegramConnect(
	stMqttSettings := stMqttSettings
);

fbMqttTelegramPingReq(
	stMqttSettings := stMqttSettings
);

fbMqttSend(
	stMqttSettings := stMqttSettings
);

(* END_ACTION *)
END_ACTION

(* POU Intern/FB_MqttTelegram_Connect_V10, ST *)
(* @NESTEDCOMMENTS := 'Yes' *)
(* @PATH := '\/_Generic\/Mqtt\/Intern' *)
(* @OBJECTFLAGS := '0, 8' *)
(* @SYMFILEFLAGS := '2048' *)
FUNCTION_BLOCK FB_MqttTelegram_Connect_V10
VAR_IN_OUT
	stMqttSettings	: ST_MqttSettings;
END_VAR
VAR
	iState 				: INT := 0;
	idLength			: INT;
	iuLength			: INT;
	ipLength			: INT;
	ipos				: INT;
	stMqttTelegram		: ST_MqttTelegram;
	fbMqttEncodeLength	: FB_Mqtt_EncodeLength_V10;
	bLength1			: BYTE;
	bLength2			: BYTE;
	bLength3			: BYTE;
	bLength4			: BYTE;
	bLengthAmount		: BYTE;
END_VAR
VAR CONSTANT
	C_STARTUP		: INT := 0;
	C_BUILD_CONNECT	: INT := 100;
	C_SEND_WAIT		: INT := 110;
	C_IDLE			: INT := 500;
END_VAR
(* @END_DECLARATION := '0' *)
CASE iState OF
	C_STARTUP:
		IF
			NOT stMqttSettings.bDisconnect
			AND NOT stMqttSettings.bError
			AND stMqttSettings.bSocketConnection
			AND stMqttSettings.bActive
		THEN
			iState := C_IDLE;
		END_IF;

